LIN {X 0,Y 229.608,Z 438.992,A -85,B 0,C 180,E1 -19914.647,E2 -19914.647} C_VEL
LIN {X 0,Y 228.927,Z 425.746,A -85,B 0,C 180,E1 -19915.956,E2 -19915.956} C_VEL
LIN {X 0,Y 227.95,Z 410.113,A -85,B 0,C 180,E1 -19917.144,E2 -19917.144} C_VEL
LIN {X 0,Y 229.155,Z 402.055,A -85,B 0,C 180,E1 -19921.424,E2 -19921.424} C_VEL
LIN {X 0,Y 230.589,Z 394.783,A -85,B 0,C 180,E1 -19925.386,E2 -19925.386} C_VEL
LIN {X 0,Y 231.878,Z 388.889,A -85,B 0,C 180,E1 -19928.622,E2 -19928.622} C_VEL
LIN {X 0,Y 231.502,Z 385.409,A -85,B 0,C 180,E1 -19930.627,E2 -19930.627} C_VEL
LIN {X 0,Y 229.924,Z 377.597,A -85,B 0,C 180,E1 -19935.329,E2 -19935.329} C_VEL
LIN {X 0,Y 228.4,Z 369.835,A -85,B 0,C 180,E1 -19940.286,E2 -19940.286} C_VEL
LIN {X 0,Y 227.949,Z 367.157,A -85,B 0,C 180,E1 -19942.123,E2 -19942.123} C_VEL
LIN {X 0,Y 227.876,Z 367.099,A -85,B 0,C 180,E1 -19946.377,E2 -19946.377} C_VEL
LIN {X 0,Y 227.915,Z 367.092,A -85,B 0,C 180,E1 -19950.437,E2 -19950.437} C_VEL
LIN {X 0,Y 227.921,Z 367.093,A -85,B 0,C 180,E1 -19954.425,E2 -19954.425} C_VEL
LIN {X 0,Y 227.939,Z 367.087,A -85,B 0,C 180,E1 -19958.285,E2 -19958.285} C_VEL
LIN {X 0,Y 228.018,Z 367.079,A -85,B 0,C 180,E1 -19963.895,E2 -19963.895} C_VEL
LIN {X 0,Y 228.049,Z 367.073,A -85,B 0,C 180,E1 -19967.542,E2 -19967.542} C_VEL
LIN {X 0,Y 228.243,Z 367.054,A -85,B 0,C 180,E1 -19971.144,E2 -19971.144} C_VEL
LIN {X 0,Y 228.308,Z 367.048,A -85,B 0,C 180,E1 -19972.927,E2 -19972.927} C_VEL
LIN {X 0,Y 228.546,Z 367.013,A -85,B 0,C 180,E1 -19978.238,E2 -19978.238} C_VEL
LIN {X 0,Y 228.547,Z 367.014,A -85,B 0,C 180,E1 -19981.762,E2 -19981.762} C_VEL
LIN {X 0,Y 228.347,Z 367.04,A -85,B 0,C 180,E1 -19987.072,E2 -19987.072} C_VEL
LIN {X 0,Y 228.158,Z 367.066,A -85,B 0,C 180,E1 -19990.651,E2 -19990.651} C_VEL
LIN {X 0,Y 228.057,Z 367.074,A -85,B 0,C 180,E1 -19994.273,E2 -19994.273} C_VEL
LIN {X 0,Y 227.999,Z 367.083,A -85,B 0,C 180,E1 -19997.954,E2 -19997.954} C_VEL
LIN {X 0,Y 227.926,Z 367.091,A -85,B 0,C 180,E1 -20002.329,E2 -20002.329} C_VEL
LIN {X 0,Y 227.939,Z 367.092,A -85,B 0,C 180,E1 -20006.603,E2 -20006.603} C_VEL
LIN {X 0,Y 227.905,Z 367.095,A -85,B 0,C 180,E1 -20010.297,E2 -20010.297} C_VEL
LIN {X 0,Y 227.886,Z 367.097,A -85,B 0,C 180,E1 -20013.719,E2 -20013.719} C_VEL
LIN {X 0,Y 227.868,Z 367.099,A -85,B 0,C 180,E1 -20018.086,E2 -20018.086} C_VEL
LIN {X 0,Y 227.834,Z 367.107,A -85,B 0,C 180,E1 -20022.242,E2 -20022.242} C_VEL
LIN {X 0,Y 227.833,Z 367.102,A -85,B 0,C 180,E1 -20025.193,E2 -20025.193} C_VEL
LIN {X 0,Y 227.824,Z 367.105,A -85,B 0,C 180,E1 -20029.624,E2 -20029.624} C_VEL
LIN {X 0,Y 227.898,Z 367.095,A -85,B 0,C 180,E1 -20034.132,E2 -20034.132} C_VEL
LIN {X 0,Y 227.872,Z 367.1,A -85,B 0,C 180,E1 -20038.379,E2 -20038.379} C_VEL
LIN {X 0,Y 227.888,Z 367.094,A -85,B 0,C 180,E1 -20042.446,E2 -20042.446} C_VEL
LIN {X 0,Y 227.915,Z 367.094,A -85,B 0,C 180,E1 -20046.368,E2 -20046.368} C_VEL
LIN {X 0,Y 227.944,Z 367.088,A -85,B 0,C 180,E1 -20050.175,E2 -20050.175} C_VEL
LIN {X 0,Y 228.059,Z 367.078,A -85,B 0,C 180,E1 -20053.898,E2 -20053.898} C_VEL
LIN {X 0,Y 228.173,Z 367.06,A -85,B 0,C 180,E1 -20059.35,E2 -20059.35} C_VEL
LIN {X 0,Y 228.361,Z 367.038,A -85,B 0,C 180,E1 -20062.929,E2 -20062.929} C_VEL
LIN {X 0,Y 228.56,Z 367.013,A -85,B 0,C 180,E1 -20068.238,E2 -20068.238} C_VEL
LIN {X 0,Y 228.557,Z 367.014,A -85,B 0,C 180,E1 -20071.762,E2 -20071.762} C_VEL
LIN {X 0,Y 228.351,Z 367.038,A -85,B 0,C 180,E1 -20077.071,E2 -20077.071} C_VEL
LIN {X 0,Y 228.16,Z 367.062,A -85,B 0,C 180,E1 -20080.65,E2 -20080.65} C_VEL
LIN {X 0,Y 228.066,Z 367.074,A -85,B 0,C 180,E1 -20084.272,E2 -20084.272} C_VEL
LIN {X 0,Y 228.004,Z 367.083,A -85,B 0,C 180,E1 -20087.953,E2 -20087.953} C_VEL
LIN {X 0,Y 227.931,Z 367.092,A -85,B 0,C 180,E1 -20092.329,E2 -20092.329} C_VEL
LIN {X 0,Y 227.942,Z 367.09,A -85,B 0,C 180,E1 -20096.602,E2 -20096.602} C_VEL
LIN {X 0,Y 227.897,Z 367.097,A -85,B 0,C 180,E1 -20100.29,E2 -20100.29} C_VEL
LIN {X 0,Y 227.889,Z 367.098,A -85,B 0,C 180,E1 -20103.717,E2 -20103.717} C_VEL
LIN {X 0,Y 227.98,Z 367.279,A -85,B 0,C 180,E1 -20106.656,E2 -20106.656} C_VEL
LIN {X 0,Y 228.218,Z 368.301,A -85,B 0,C 180,E1 -20106.956,E2 -20106.956} C_VEL
LIN {X 0,Y 231.872,Z 380.761,A -85,B 0,C 180,E1 -20108.691,E2 -20108.691} C_VEL
LIN {X 0,Y 234.923,Z 392.226,A -85,B 0,C 180,E1 -20110.589,E2 -20110.589} C_VEL
LIN {X 0,Y 235.363,Z 394.934,A -85,B 0,C 180,E1 -20111.065,E2 -20111.065} C_VEL
LIN {X 0,Y 233.758,Z 406.693,A -85,B 0,C 180,E1 -20113.19,E2 -20113.19} C_VEL
LIN {X 0,Y 232.42,Z 416.268,A -85,B 0,C 180,E1 -20115.328,E2 -20115.328} C_VEL
LIN {X 0,Y 231,Z 425.883,A -85,B 0,C 180,E1 -20117.984,E2 -20117.984} C_VEL
LIN {X 0,Y 229.917,Z 433.61,A -85,B 0,C 180,E1 -20120.634,E2 -20120.634} C_VEL
LIN {X 0,Y 229.046,Z 440.448,A -85,B 0,C 180,E1 -20123.582,E2 -20123.582} C_VEL
LIN {X 0,Y 228.563,Z 445.529,A -85,B 0,C 180,E1 -20126.394,E2 -20126.394} C_VEL
LIN {X 0,Y 228.351,Z 449.786,A -85,B 0,C 180,E1 -20129.512,E2 -20129.512} C_VEL
LIN {X 0,Y 228.594,Z 453.024,A -85,B 0,C 180,E1 -20133.071,E2 -20133.071} C_VEL
LIN {X 0,Y 229.502,Z 454.674,A -85,B 0,C 180,E1 -20136.731,E2 -20136.731} C_VEL
LIN {X 0,Y 230.188,Z 454.837,A -85,B 0,C 180,E1 -20138.507,E2 -20138.507} C_VEL
LIN {X 0,Y 231.096,Z 454.553,A -85,B 0,C 180,E1 -20140.516,E2 -20140.516} C_VEL
LIN {X 0,Y 232.177,Z 453.845,A -85,B 0,C 180,E1 -20142.38,E2 -20142.38} C_VEL
LIN {X 0,Y 233.489,Z 452.509,A -85,B 0,C 180,E1 -20144.402,E2 -20144.402} C_VEL
LIN {X 0,Y 235.627,Z 449.858,A -85,B 0,C 180,E1 -20147.074,E2 -20147.074} C_VEL
LIN {X 0,Y 238.305,Z 445.922,A -85,B 0,C 180,E1 -20149.808,E2 -20149.808} C_VEL
LIN {X 0,Y 241.533,Z 440.446,A -85,B 0,C 180,E1 -20152.61,E2 -20152.61} C_VEL
LIN {X 0,Y 245.371,Z 433.011,A -85,B 0,C 180,E1 -20155.442,E2 -20155.442} C_VEL
LIN {X 0,Y 248.658,Z 425.827,A -85,B 0,C 180,E1 -20157.57,E2 -20157.57} C_VEL
LIN {X 0,Y 251.387,Z 419.09,A -85,B 0,C 180,E1 -20159.199,E2 -20159.199} C_VEL
LIN {X 0,Y 251.425,Z 416.583,A -85,B 0,C 180,E1 -20160,E2 -20160} C_VEL
LIN {X 0,Y 249.947,Z 407.014,A -85,B 0,C 180,E1 -20163.224,E2 -20163.224} C_VEL
LIN {X 0,Y 248.68,Z 402.352,A -85,B 0,C 180,E1 -20164.864,E2 -20164.864} C_VEL
LIN {X 0,Y 245.143,Z 393.716,A -85,B 0,C 180,E1 -20168.242,E2 -20168.242} C_VEL
LIN {X 0,Y 241.797,Z 387.198,A -85,B 0,C 180,E1 -20171.14,E2 -20171.14} C_VEL
LIN {X 0,Y 239.703,Z 383.456,A -85,B 0,C 180,E1 -20172.976,E2 -20172.976} C_VEL
LIN {X 0,Y 236.75,Z 379.72,A -85,B 0,C 180,E1 -20175.496,E2 -20175.496} C_VEL
LIN {X 0,Y 234.248,Z 377.714,A -85,B 0,C 180,E1 -20177.685,E2 -20177.685} C_VEL
LIN {X 0,Y 233.353,Z 376.567,A -85,B 0,C 180,E1 -20178.663,E2 -20178.663} C_VEL
LIN {X 0,Y 230.291,Z 375.175,A -85,B 0,C 180,E1 -20182.071,E2 -20182.071} C_VEL
LIN {X 0,Y 229.631,Z 374.388,A -85,B 0,C 180,E1 -20183.445,E2 -20183.445} C_VEL
LIN {X 0,Y 229.685,Z 374.739,A -85,B 0,C 180,E1 -20185.365,E2 -20185.365} C_VEL
LIN {X 0,Y 229.986,Z 375.936,A -85,B 0,C 180,E1 -20187.604,E2 -20187.604} C_VEL
LIN {X 0,Y 230.436,Z 378.369,A -85,B 0,C 180,E1 -20191.357,E2 -20191.357} C_VEL
LIN {X 0,Y 231.054,Z 381.457,A -85,B 0,C 180,E1 -20195.305,E2 -20195.305} C_VEL
LIN {X 0,Y 231.986,Z 385.695,A -85,B 0,C 180,E1 -20199.807,E2 -20199.807} C_VEL
LIN {X 0,Y 232.582,Z 388.031,A -85,B 0,C 180,E1 -20201.359,E2 -20201.359} C_VEL
LIN {X 0,Y 235.887,Z 395.137,A -85,B 0,C 180,E1 -20204.588,E2 -20204.588} C_VEL
LIN {X 0,Y 237.313,Z 397.724,A -85,B 0,C 180,E1 -20205.7,E2 -20205.7} C_VEL
LIN {X 0,Y 239.366,Z 402.878,A -85,B 0,C 180,E1 -20207.386,E2 -20207.386} C_VEL
LIN {X 0,Y 240.173,Z 404.323,A -85,B 0,C 180,E1 -20207.949,E2 -20207.949} C_VEL
LIN {X 0,Y 241.673,Z 410.353,A -85,B 0,C 180,E1 -20209.395,E2 -20209.395} C_VEL
LIN {X 0,Y 242.991,Z 419.215,A -85,B 0,C 180,E1 -20211.252,E2 -20211.252} C_VEL
LIN {X 0,Y 243.153,Z 423.985,A -85,B 0,C 180,E1 -20212.075,E2 -20212.075} C_VEL
LIN {X 0,Y 242.458,Z 429.111,A -85,B 0,C 180,E1 -20212.768,E2 -20212.768} C_VEL
LIN {X 0,Y 239.789,Z 439.501,A -85,B 0,C 180,E1 -20214.065,E2 -20214.065} C_VEL
LIN {X 0,Y 238.717,Z 444.414,A -85,B 0,C 180,E1 -20214.849,E2 -20214.849} C_VEL
LIN {X 0,Y 238.543,Z 445.927,A -85,B 0,C 180,E1 -20215.153,E2 -20215.153} C_VEL
LIN {X 0,Y 237.13,Z 458.322,A -85,B 0,C 180,E1 -20217.76,E2 -20217.76} C_VEL
LIN {X 0,Y 234.95,Z 468.801,A -85,B 0,C 180,E1 -20220.166,E2 -20220.166} C_VEL
LIN {X 0,Y 231.595,Z 479.491,A -85,B 0,C 180,E1 -20222.923,E2 -20222.923} C_VEL
LIN {X 0,Y 228.665,Z 487.706,A -85,B 0,C 180,E1 -20225.486,E2 -20225.486} C_VEL
LIN {X 0,Y 225.158,Z 495.637,A -85,B 0,C 180,E1 -20228.485,E2 -20228.485} C_VEL
LIN {X 0,Y 222.418,Z 502.006,A -85,B 0,C 180,E1 -20231.58,E2 -20231.58} C_VEL
LIN {X 0,Y 220.511,Z 507.656,A -85,B 0,C 180,E1 -20235.229,E2 -20235.229} C_VEL
LIN {X 0,Y 219.511,Z 511.634,A -85,B 0,C 180,E1 -20238.925,E2 -20238.925} C_VEL
LIN {X 0,Y 219.626,Z 514.192,A -85,B 0,C 180,E1 -20242.747,E2 -20242.747} C_VEL
LIN {X 0,Y 219.956,Z 514.809,A -85,B 0,C 180,E1 -20244.5,E2 -20244.5} C_VEL
LIN {X 0,Y 220.893,Z 514.907,A -85,B 0,C 180,E1 -20248.177,E2 -20248.177} C_VEL
LIN {X 0,Y 221.448,Z 514.346,A -85,B 0,C 180,E1 -20250,E2 -20250} C_VEL
LIN {X 0,Y 221.043,Z 513.169,A -85,B 0,C 180,E1 -20251.822,E2 -20251.822} C_VEL
LIN {X 0,Y 220.637,Z 510.508,A -85,B 0,C 180,E1 -20254.567,E2 -20254.567} C_VEL
LIN {X 0,Y 220.226,Z 506.669,A -85,B 0,C 180,E1 -20257.334,E2 -20257.334} C_VEL
LIN {X 0,Y 220.1,Z 501.587,A -85,B 0,C 180,E1 -20260.115,E2 -20260.115} C_VEL
LIN {X 0,Y 220.464,Z 495.155,A -85,B 0,C 180,E1 -20262.894,E2 -20262.894} C_VEL
LIN {X 0,Y 221.315,Z 487.153,A -85,B 0,C 180,E1 -20265.659,E2 -20265.659} C_VEL
LIN {X 0,Y 222.477,Z 479.009,A -85,B 0,C 180,E1 -20267.938,E2 -20267.938} C_VEL
LIN {X 0,Y 223.11,Z 473.256,A -85,B 0,C 180,E1 -20269.296,E2 -20269.296} C_VEL
LIN {X 0,Y 223.125,Z 462.474,A -85,B 0,C 180,E1 -20271.479,E2 -20271.479} C_VEL
LIN {X 0,Y 222.936,Z 451.084,A -85,B 0,C 180,E1 -20273.358,E2 -20273.358} C_VEL
LIN {X 0,Y 222.547,Z 438.854,A -85,B 0,C 180,E1 -20274.984,E2 -20274.984} C_VEL
LIN {X 0,Y 221.982,Z 426.264,A -85,B 0,C 180,E1 -20276.31,E2 -20276.31} C_VEL
LIN {X 0,Y 221.011,Z 410.739,A -85,B 0,C 180,E1 -20277.512,E2 -20277.512} C_VEL
LIN {X 0,Y 220.986,Z 408.993,A -85,B 0,C 180,E1 -20277.72,E2 -20277.72} C_VEL
LIN {X 0,Y 222.797,Z 398.631,A -85,B 0,C 180,E1 -20283.505,E2 -20283.505} C_VEL
LIN {X 0,Y 224.768,Z 389.696,A -85,B 0,C 180,E1 -20288.584,E2 -20288.584} C_VEL
LIN {X 0,Y 224.454,Z 386.287,A -85,B 0,C 180,E1 -20290.598,E2 -20290.598} C_VEL
LIN {X 0,Y 223.029,Z 379.316,A -85,B 0,C 180,E1 -20294.918,E2 -20294.918} C_VEL
LIN {X 0,Y 221.608,Z 372.183,A -85,B 0,C 180,E1 -20299.562,E2 -20299.562} C_VEL
LIN {X 0,Y 220.874,Z 368.016,A -85,B 0,C 180,E1 -20302.545,E2 -20302.545} C_VEL
LIN {X 0,Y 220.814,Z 367.981,A -85,B 0,C 180,E1 -20307.243,E2 -20307.243} C_VEL
LIN {X 0,Y 220.833,Z 367.976,A -85,B 0,C 180,E1 -20311.486,E2 -20311.486} C_VEL
LIN {X 0,Y 220.858,Z 367.972,A -85,B 0,C 180,E1 -20315.564,E2 -20315.564} C_VEL
LIN {X 0,Y 220.87,Z 367.971,A -85,B 0,C 180,E1 -20319.512,E2 -20319.512} C_VEL
LIN {X 0,Y 220.974,Z 367.958,A -85,B 0,C 180,E1 -20323.367,E2 -20323.367} C_VEL
LIN {X 0,Y 221.056,Z 367.947,A -85,B 0,C 180,E1 -20329.003,E2 -20329.003} C_VEL
LIN {X 0,Y 221.242,Z 367.927,A -85,B 0,C 180,E1 -20332.7,E2 -20332.7} C_VEL
LIN {X 0,Y 221.504,Z 367.89,A -85,B 0,C 180,E1 -20338.182,E2 -20338.182} C_VEL
LIN {X 0,Y 221.505,Z 367.891,A -85,B 0,C 180,E1 -20341.818,E2 -20341.818} C_VEL
LIN {X 0,Y 221.283,Z 367.919,A -85,B 0,C 180,E1 -20347.299,E2 -20347.299} C_VEL
LIN {X 0,Y 221.107,Z 367.942,A -85,B 0,C 180,E1 -20350.994,E2 -20350.994} C_VEL
LIN {X 0,Y 221.011,Z 367.957,A -85,B 0,C 180,E1 -20356.63,E2 -20356.63} C_VEL
LIN {X 0,Y 220.888,Z 367.969,A -85,B 0,C 180,E1 -20360.487,E2 -20360.487} C_VEL
LIN {X 0,Y 220.863,Z 367.974,A -85,B 0,C 180,E1 -20364.435,E2 -20364.435} C_VEL
LIN {X 0,Y 220.833,Z 367.976,A -85,B 0,C 180,E1 -20368.514,E2 -20368.514} C_VEL
LIN {X 0,Y 220.821,Z 367.978,A -85,B 0,C 180,E1 -20372.755,E2 -20372.755} C_VEL
LIN {X 0,Y 220.836,Z 367.973,A -85,B 0,C 180,E1 -20377.289,E2 -20377.289} C_VEL
LIN {X 0,Y 220.835,Z 367.977,A -85,B 0,C 180,E1 -20380.202,E2 -20380.202} C_VEL
LIN {X 0,Y 220.777,Z 367.983,A -85,B 0,C 180,E1 -20384.453,E2 -20384.453} C_VEL
LIN {X 0,Y 220.768,Z 367.984,A -85,B 0,C 180,E1 -20388.048,E2 -20388.048} C_VEL
LIN {X 0,Y 220.823,Z 367.975,A -85,B 0,C 180,E1 -20392.794,E2 -20392.794} C_VEL
LIN {X 0,Y 220.823,Z 367.976,A -85,B 0,C 180,E1 -20397.246,E2 -20397.246} C_VEL
LIN {X 0,Y 220.838,Z 367.975,A -85,B 0,C 180,E1 -20401.487,E2 -20401.487} C_VEL
LIN {X 0,Y 220.868,Z 367.972,A -85,B 0,C 180,E1 -20405.566,E2 -20405.566} C_VEL
LIN {X 0,Y 220.894,Z 367.969,A -85,B 0,C 180,E1 -20409.515,E2 -20409.515} C_VEL
LIN {X 0,Y 221.018,Z 367.952,A -85,B 0,C 180,E1 -20413.371,E2 -20413.371} C_VEL
LIN {X 0,Y 221.118,Z 367.938,A -85,B 0,C 180,E1 -20419.006,E2 -20419.006} C_VEL
LIN {X 0,Y 221.314,Z 367.915,A -85,B 0,C 180,E1 -20422.703,E2 -20422.703} C_VEL
LIN {X 0,Y 221.517,Z 367.89,A -85,B 0,C 180,E1 -20428.182,E2 -20428.182} C_VEL
LIN {X 0,Y 221.515,Z 367.891,A -85,B 0,C 180,E1 -20431.818,E2 -20431.818} C_VEL
LIN {X 0,Y 221.286,Z 367.919,A -85,B 0,C 180,E1 -20437.298,E2 -20437.298} C_VEL
LIN {X 0,Y 221.108,Z 367.942,A -85,B 0,C 180,E1 -20440.994,E2 -20440.994} C_VEL
LIN {X 0,Y 221.018,Z 367.952,A -85,B 0,C 180,E1 -20446.629,E2 -20446.629} C_VEL
LIN {X 0,Y 220.894,Z 367.968,A -85,B 0,C 180,E1 -20450.485,E2 -20450.485} C_VEL
LIN {X 0,Y 220.868,Z 367.971,A -85,B 0,C 180,E1 -20454.434,E2 -20454.434} C_VEL
LIN {X 0,Y 220.827,Z 367.977,A -85,B 0,C 180,E1 -20458.514,E2 -20458.514} C_VEL
LIN {X 0,Y 220.822,Z 367.979,A -85,B 0,C 180,E1 -20462.754,E2 -20462.754} C_VEL
LIN {X 0,Y 220.938,Z 368.197,A -85,B 0,C 180,E1 -20466.189,E2 -20466.189} C_VEL
LIN {X 0,Y 221.315,Z 369.606,A -85,B 0,C 180,E1 -20466.541,E2 -20466.541} C_VEL
LIN {X 0,Y 225.032,Z 382.472,A -85,B 0,C 180,E1 -20468.391,E2 -20468.391} C_VEL
LIN {X 0,Y 228.05,Z 393.725,A -85,B 0,C 180,E1 -20470.328,E2 -20470.328} C_VEL
LIN {X 0,Y 228.436,Z 396.031,A -85,B 0,C 180,E1 -20470.746,E2 -20470.746} C_VEL
LIN {X 0,Y 227,Z 406.259,A -85,B 0,C 180,E1 -20472.623,E2 -20472.623} C_VEL
LIN {X 0,Y 225.346,Z 417.549,A -85,B 0,C 180,E1 -20475.199,E2 -20475.199} C_VEL
LIN {X 0,Y 224.07,Z 426.024,A -85,B 0,C 180,E1 -20477.596,E2 -20477.596} C_VEL
LIN {X 0,Y 222.908,Z 434.092,A -85,B 0,C 180,E1 -20480.41,E2 -20480.41} C_VEL
LIN {X 0,Y 222.102,Z 440.214,A -85,B 0,C 180,E1 -20483.043,E2 -20483.043} C_VEL
LIN {X 0,Y 221.481,Z 446.408,A -85,B 0,C 180,E1 -20486.444,E2 -20486.444} C_VEL
LIN {X 0,Y 221.305,Z 450.496,A -85,B 0,C 180,E1 -20489.462,E2 -20489.462} C_VEL
LIN {X 0,Y 221.488,Z 453.578,A -85,B 0,C 180,E1 -20492.678,E2 -20492.678} C_VEL
LIN {X 0,Y 222.372,Z 455.557,A -85,B 0,C 180,E1 -20496.422,E2 -20496.422} C_VEL
LIN {X 0,Y 223.72,Z 455.93,A -85,B 0,C 180,E1 -20499.784,E2 -20499.784} C_VEL
LIN {X 0,Y 224.754,Z 455.531,A -85,B 0,C 180,E1 -20501.778,E2 -20501.778} C_VEL
LIN {X 0,Y 226.352,Z 454.314,A -85,B 0,C 180,E1 -20504.258,E2 -20504.258} C_VEL
LIN {X 0,Y 229.023,Z 451.371,A -85,B 0,C 180,E1 -20507.596,E2 -20507.596} C_VEL
LIN {X 0,Y 231.875,Z 447.588,A -85,B 0,C 180,E1 -20510.404,E2 -20510.404} C_VEL
LIN {X 0,Y 235.101,Z 442.579,A -85,B 0,C 180,E1 -20513.133,E2 -20513.133} C_VEL
LIN {X 0,Y 238.723,Z 436.177,A -85,B 0,C 180,E1 -20515.768,E2 -20515.768} C_VEL
LIN {X 0,Y 242.764,Z 428.059,A -85,B 0,C 180,E1 -20518.341,E2 -20518.341} C_VEL
LIN {X 0,Y 245.655,Z 421.564,A -85,B 0,C 180,E1 -20520,E2 -20520} C_VEL
LIN {X 0,Y 245.225,Z 415.957,A -85,B 0,C 180,E1 -20522.053,E2 -20522.053} C_VEL
LIN {X 0,Y 244.303,Z 409.245,A -85,B 0,C 180,E1 -20524.465,E2 -20524.465} C_VEL
LIN {X 0,Y 242.566,Z 403.762,A -85,B 0,C 180,E1 -20526.655,E2 -20526.655} C_VEL
LIN {X 0,Y 239.933,Z 396.884,A -85,B 0,C 180,E1 -20529.61,E2 -20529.61} C_VEL
LIN {X 0,Y 236.466,Z 389.951,A -85,B 0,C 180,E1 -20533.156,E2 -20533.156} C_VEL
LIN {X 0,Y 233.769,Z 386.071,A -85,B 0,C 180,E1 -20535.841,E2 -20535.841} C_VEL
LIN {X 0,Y 230.623,Z 383.152,A -85,B 0,C 180,E1 -20539.149,E2 -20539.149} C_VEL
LIN {X 0,Y 227.995,Z 381.679,A -85,B 0,C 180,E1 -20542.633,E2 -20542.633} C_VEL
LIN {X 0,Y 227.528,Z 381.149,A -85,B 0,C 180,E1 -20543.675,E2 -20543.675} C_VEL
LIN {X 0,Y 226.051,Z 381.62,A -85,B 0,C 180,E1 -20547.105,E2 -20547.105} C_VEL
LIN {X 0,Y 225.556,Z 383.422,A -85,B 0,C 180,E1 -20551.095,E2 -20551.095} C_VEL
LIN {X 0,Y 226.222,Z 386.236,A -85,B 0,C 180,E1 -20554.588,E2 -20554.588} C_VEL
LIN {X 0,Y 228.937,Z 391.93,A -85,B 0,C 180,E1 -20559.427,E2 -20559.427} C_VEL
LIN {X 0,Y 230.112,Z 394.682,A -85,B 0,C 180,E1 -20560.976,E2 -20560.976} C_VEL
LIN {X 0,Y 232.854,Z 401.033,A -85,B 0,C 180,E1 -20563.963,E2 -20563.963} C_VEL
LIN {X 0,Y 233.668,Z 402.418,A -85,B 0,C 180,E1 -20564.675,E2 -20564.675} C_VEL
LIN {X 0,Y 235.763,Z 408.322,A -85,B 0,C 180,E1 -20566.717,E2 -20566.717} C_VEL
LIN {X 0,Y 236.66,Z 410.544,A -85,B 0,C 180,E1 -20567.509,E2 -20567.509} C_VEL
LIN {X 0,Y 237.395,Z 415.062,A -85,B 0,C 180,E1 -20568.6,E2 -20568.6} C_VEL
LIN {X 0,Y 238.328,Z 423.701,A -85,B 0,C 180,E1 -20570.517,E2 -20570.517} C_VEL
LIN {X 0,Y 238.854,Z 436.554,A -85,B 0,C 180,E1 -20573.205,E2 -20573.205} C_VEL
LIN {X 0,Y 238.543,Z 445.927,A -85,B 0,C 180,E1 -20575.153,E2 -20575.153} C_VEL
LIN {X 0,Y 237.596,Z 450.708,A -85,B 0,C 180,E1 -20576.014,E2 -20576.014} C_VEL
LIN {X 0,Y 235.73,Z 455.509,A -85,B 0,C 180,E1 -20576.759,E2 -20576.759} C_VEL
LIN {X 0,Y 231.021,Z 464.66,A -85,B 0,C 180,E1 -20578.239,E2 -20578.239} C_VEL
LIN {X 0,Y 229.077,Z 468.943,A -85,B 0,C 180,E1 -20579.133,E2 -20579.133} C_VEL
LIN {X 0,Y 228.619,Z 470.288,A -85,B 0,C 180,E1 -20579.468,E2 -20579.468} C_VEL
LIN {X 0,Y 225.282,Z 479.825,A -85,B 0,C 180,E1 -20582.1,E2 -20582.1} C_VEL
LIN {X 0,Y 221.657,Z 488.946,A -85,B 0,C 180,E1 -20585.159,E2 -20585.159} C_VEL
LIN {X 0,Y 218.079,Z 496.39,A -85,B 0,C 180,E1 -20588.247,E2 -20588.247} C_VEL
LIN {X 0,Y 215.056,Z 503.063,A -85,B 0,C 180,E1 -20591.914,E2 -20591.914} C_VEL
LIN {X 0,Y 213.215,Z 508.098,A -85,B 0,C 180,E1 -20595.688,E2 -20595.688} C_VEL
LIN {X 0,Y 212.502,Z 510.799,A -85,B 0,C 180,E1 -20598.555,E2 -20598.555} C_VEL
LIN {X 0,Y 212.537,Z 513.13,A -85,B 0,C 180,E1 -20602.4,E2 -20602.4} C_VEL
LIN {X 0,Y 212.886,Z 513.711,A -85,B 0,C 180,E1 -20604.316,E2 -20604.316} C_VEL
LIN {X 0,Y 213.845,Z 513.703,A -85,B 0,C 180,E1 -20608.117,E2 -20608.117} C_VEL
LIN {X 0,Y 214.431,Z 513.093,A -85,B 0,C 180,E1 -20610,E2 -20610} C_VEL
LIN {X 0,Y 214.039,Z 511.812,A -85,B 0,C 180,E1 -20611.882,E2 -20611.882} C_VEL
LIN {X 0,Y 213.613,Z 509.022,A -85,B 0,C 180,E1 -20614.718,E2 -20614.718} C_VEL
LIN {X 0,Y 213.175,Z 505.032,A -85,B 0,C 180,E1 -20617.578,E2 -20617.578} C_VEL
LIN {X 0,Y 213.166,Z 498.831,A -85,B 0,C 180,E1 -20620.928,E2 -20620.928} C_VEL
LIN {X 0,Y 213.61,Z 491.961,A -85,B 0,C 180,E1 -20623.8,E2 -20623.8} C_VEL
LIN {X 0,Y 214.676,Z 483.403,A -85,B 0,C 180,E1 -20626.645,E2 -20626.645} C_VEL
LIN {X 0,Y 215.976,Z 474.691,A -85,B 0,C 180,E1 -20628.99,E2 -20628.99} C_VEL
LIN {X 0,Y 216.065,Z 464.592,A -85,B 0,C 180,E1 -20631.214,E2 -20631.214} C_VEL
LIN {X 0,Y 215.905,Z 452.698,A -85,B 0,C 180,E1 -20633.351,E2 -20633.351} C_VEL
LIN {X 0,Y 215.644,Z 440.924,A -85,B 0,C 180,E1 -20635.066,E2 -20635.066} C_VEL
LIN {X 0,Y 215.114,Z 427.854,A -85,B 0,C 180,E1 -20636.563,E2 -20636.563} C_VEL
LIN {X 0,Y 214.351,Z 414.249,A -85,B 0,C 180,E1 -20637.746,E2 -20637.746} C_VEL
LIN {X 0,Y 214.006,Z 408.243,A -85,B 0,C 180,E1 -20638.214,E2 -20638.214} C_VEL
LIN {X 0,Y 215.331,Z 400.48,A -85,B 0,C 180,E1 -20642.647,E2 -20642.647} C_VEL
LIN {X 0,Y 217.355,Z 391.513,A -85,B 0,C 180,E1 -20647.903,E2 -20647.903} C_VEL
LIN {X 0,Y 217.723,Z 389.305,A -85,B 0,C 180,E1 -20649.221,E2 -20649.221} C_VEL
LIN {X 0,Y 216.625,Z 383.378,A -85,B 0,C 180,E1 -20652.944,E2 -20652.944} C_VEL
LIN {X 0,Y 215.095,Z 375.852,A -85,B 0,C 180,E1 -20657.885,E2 -20657.885} C_VEL
LIN {X 0,Y 213.83,Z 368.918,A -85,B 0,C 180,E1 -20662.769,E2 -20662.769} C_VEL
LIN {X 0,Y 213.754,Z 368.858,A -85,B 0,C 180,E1 -20666.017,E2 -20666.017} C_VEL
LIN {X 0,Y 213.777,Z 368.853,A -85,B 0,C 180,E1 -20670.453,E2 -20670.453} C_VEL
LIN {X 0,Y 213.794,Z 368.853,A -85,B 0,C 180,E1 -20674.701,E2 -20674.701} C_VEL
LIN {X 0,Y 213.792,Z 368.851,A -85,B 0,C 180,E1 -20678.801,E2 -20678.801} C_VEL
LIN {X 0,Y 213.888,Z 368.843,A -85,B 0,C 180,E1 -20682.799,E2 -20682.799} C_VEL
LIN {X 0,Y 213.929,Z 368.831,A -85,B 0,C 180,E1 -20686.705,E2 -20686.705} C_VEL
LIN {X 0,Y 214.12,Z 368.811,A -85,B 0,C 180,E1 -20690.554,E2 -20690.554} C_VEL
LIN {X 0,Y 214.087,Z 368.816,A -85,B 0,C 180,E1 -20694.348,E2 -20694.348} C_VEL
LIN {X 0,Y 214.437,Z 368.77,A -85,B 0,C 180,E1 -20698.122,E2 -20698.122} C_VEL
LIN {X 0,Y 214.544,Z 368.758,A -85,B 0,C 180,E1 -20700,E2 -20700} C_VEL
LIN {X 0,Y 214.438,Z 368.772,A -85,B 0,C 180,E1 -20701.878,E2 -20701.878} C_VEL
LIN {X 0,Y 214.221,Z 368.798,A -85,B 0,C 180,E1 -20707.541,E2 -20707.541} C_VEL
LIN {X 0,Y 214.04,Z 368.821,A -85,B 0,C 180,E1 -20711.362,E2 -20711.362} C_VEL
LIN {X 0,Y 213.927,Z 368.835,A -85,B 0,C 180,E1 -20715.237,E2 -20715.237} C_VEL
LIN {X 0,Y 213.835,Z 368.847,A -85,B 0,C 180,E1 -20719.188,E2 -20719.188} C_VEL
LIN {X 0,Y 213.843,Z 368.845,A -85,B 0,C 180,E1 -20723.227,E2 -20723.227} C_VEL
LIN {X 0,Y 213.826,Z 368.848,A -85,B 0,C 180,E1 -20727.45,E2 -20727.45} C_VEL
LIN {X 0,Y 213.776,Z 368.853,A -85,B 0,C 180,E1 -20731.736,E2 -20731.736} C_VEL
LIN {X 0,Y 213.751,Z 368.859,A -85,B 0,C 180,E1 -20736.287,E2 -20736.287} C_VEL
LIN {X 0,Y 213.75,Z 368.858,A -85,B 0,C 180,E1 -20740.869,E2 -20740.869} C_VEL
LIN {X 0,Y 213.746,Z 368.859,A -85,B 0,C 180,E1 -20743.669,E2 -20743.669} C_VEL
LIN {X 0,Y 213.71,Z 368.862,A -85,B 0,C 180,E1 -20748.876,E2 -20748.876} C_VEL
LIN {X 0,Y 213.747,Z 368.858,A -85,B 0,C 180,E1 -20753.713,E2 -20753.713} C_VEL
LIN {X 0,Y 213.779,Z 368.856,A -85,B 0,C 180,E1 -20758.265,E2 -20758.265} C_VEL
LIN {X 0,Y 213.826,Z 368.845,A -85,B 0,C 180,E1 -20762.604,E2 -20762.604} C_VEL
LIN {X 0,Y 213.853,Z 368.845,A -85,B 0,C 180,E1 -20766.953,E2 -20766.953} C_VEL
LIN {X 0,Y 213.945,Z 368.832,A -85,B 0,C 180,E1 -20772.804,E2 -20772.804} C_VEL
LIN {X 0,Y 213.982,Z 368.828,A -85,B 0,C 180,E1 -20776.709,E2 -20776.709} C_VEL
LIN {X 0,Y 214.198,Z 368.8,A -85,B 0,C 180,E1 -20780.558,E2 -20780.558} C_VEL
LIN {X 0,Y 214.25,Z 368.796,A -85,B 0,C 180,E1 -20782.461,E2 -20782.461} C_VEL
LIN {X 0,Y 214.451,Z 368.771,A -85,B 0,C 180,E1 -20788.122,E2 -20788.122} C_VEL
LIN {X 0,Y 214.557,Z 368.758,A -85,B 0,C 180,E1 -20790,E2 -20790} C_VEL
LIN {X 0,Y 214.449,Z 368.771,A -85,B 0,C 180,E1 -20791.878,E2 -20791.878} C_VEL
LIN {X 0,Y 214.224,Z 368.801,A -85,B 0,C 180,E1 -20797.54,E2 -20797.54} C_VEL
LIN {X 0,Y 214.025,Z 368.823,A -85,B 0,C 180,E1 -20801.363,E2 -20801.363} C_VEL
LIN {X 0,Y 213.936,Z 368.838,A -85,B 0,C 180,E1 -20805.236,E2 -20805.236} C_VEL
LIN {X 0,Y 213.869,Z 368.846,A -85,B 0,C 180,E1 -20809.184,E2 -20809.184} C_VEL
LIN {X 0,Y 213.848,Z 368.848,A -85,B 0,C 180,E1 -20813.226,E2 -20813.226} C_VEL
LIN {X 0,Y 213.829,Z 368.85,A -85,B 0,C 180,E1 -20817.449,E2 -20817.449} C_VEL
LIN {X 0,Y 213.769,Z 368.858,A -85,B 0,C 180,E1 -20821.736,E2 -20821.736} C_VEL
LIN {X 0,Y 213.868,Z 369.06,A -85,B 0,C 180,E1 -20825.672,E2 -20825.672} C_VEL
LIN {X 0,Y 214.114,Z 370.059,A -85,B 0,C 180,E1 -20825.978,E2 -20825.978} C_VEL
LIN {X 0,Y 217.996,Z 383.346,A -85,B 0,C 180,E1 -20827.965,E2 -20827.965} C_VEL
LIN {X 0,Y 221.115,Z 395.078,A -85,B 0,C 180,E1 -20830.057,E2 -20830.057} C_VEL
LIN {X 0,Y 221.478,Z 396.873,A -85,B 0,C 180,E1 -20830.397,E2 -20830.397} C_VEL
LIN {X 0,Y 219.996,Z 407.293,A -85,B 0,C 180,E1 -20832.369,E2 -20832.369} C_VEL
LIN {X 0,Y 218.367,Z 418.19,A -85,B 0,C 180,E1 -20834.923,E2 -20834.923} C_VEL
LIN {X 0,Y 216.859,Z 427.936,A -85,B 0,C 180,E1 -20837.786,E2 -20837.786} C_VEL
LIN {X 0,Y 215.729,Z 435.546,A -85,B 0,C 180,E1 -20840.559,E2 -20840.559} C_VEL
LIN {X 0,Y 214.964,Z 441.792,A -85,B 0,C 180,E1 -20843.369,E2 -20843.369} C_VEL
LIN {X 0,Y 214.444,Z 446.742,A -85,B 0,C 180,E1 -20846.142,E2 -20846.142} C_VEL
LIN {X 0,Y 214.241,Z 451.316,A -85,B 0,C 180,E1 -20849.52,E2 -20849.52} C_VEL
LIN {X 0,Y 214.444,Z 454.361,A -85,B 0,C 180,E1 -20852.689,E2 -20852.689} C_VEL
LIN {X 0,Y 215.222,Z 456.387,A -85,B 0,C 180,E1 -20856.107,E2 -20856.107} C_VEL
LIN {X 0,Y 216.808,Z 457.086,A -85,B 0,C 180,E1 -20860.057,E2 -20860.057} C_VEL
LIN {X 0,Y 219.194,Z 455.989,A -85,B 0,C 180,E1 -20864.125,E2 -20864.125} C_VEL
LIN {X 0,Y 221.572,Z 453.852,A -85,B 0,C 180,E1 -20867.172,E2 -20867.172} C_VEL
LIN {X 0,Y 224.414,Z 450.61,A -85,B 0,C 180,E1 -20870.082,E2 -20870.082} C_VEL
LIN {X 0,Y 227.74,Z 446.143,A -85,B 0,C 180,E1 -20872.909,E2 -20872.909} C_VEL
LIN {X 0,Y 231.389,Z 440.447,A -85,B 0,C 180,E1 -20875.646,E2 -20875.646} C_VEL
LIN {X 0,Y 235.506,Z 433.15,A -85,B 0,C 180,E1 -20878.29,E2 -20878.29} C_VEL
LIN {X 0,Y 239.494,Z 425.126,A -85,B 0,C 180,E1 -20880.563,E2 -20880.563} C_VEL
LIN {X 0,Y 239.894,Z 424.111,A -85,B 0,C 180,E1 -20880.839,E2 -20880.839} C_VEL
LIN {X 0,Y 239.375,Z 415.707,A -85,B 0,C 180,E1 -20884.125,E2 -20884.125} C_VEL
LIN {X 0,Y 238.315,Z 410.413,A -85,B 0,C 180,E1 -20886.314,E2 -20886.314} C_VEL
LIN {X 0,Y 235.474,Z 401.735,A -85,B 0,C 180,E1 -20890.316,E2 -20890.316} C_VEL
LIN {X 0,Y 232.489,Z 395.187,A -85,B 0,C 180,E1 -20893.995,E2 -20893.995} C_VEL
LIN {X 0,Y 230.833,Z 392.59,A -85,B 0,C 180,E1 -20895.904,E2 -20895.904} C_VEL
LIN {X 0,Y 227.515,Z 389.609,A -85,B 0,C 180,E1 -20899.864,E2 -20899.864} C_VEL
LIN {X 0,Y 225.208,Z 387.932,A -85,B 0,C 180,E1 -20903.934,E2 -20903.934} C_VEL
LIN {X 0,Y 224.273,Z 388.149,A -85,B 0,C 180,E1 -20906.022,E2 -20906.022} C_VEL
LIN {X 0,Y 223.526,Z 389.789,A -85,B 0,C 180,E1 -20910.203,E2 -20910.203} C_VEL
LIN {X 0,Y 223.613,Z 391.144,A -85,B 0,C 180,E1 -20912.296,E2 -20912.296} C_VEL
LIN {X 0,Y 224.873,Z 395.2,A -85,B 0,C 180,E1 -20916.428,E2 -20916.428} C_VEL
LIN {X 0,Y 226.906,Z 399.457,A -85,B 0,C 180,E1 -20919.745,E2 -20919.745} C_VEL
LIN {X 0,Y 229.482,Z 406.676,A -85,B 0,C 180,E1 -20923.268,E2 -20923.268} C_VEL
LIN {X 0,Y 230.166,Z 407.946,A -85,B 0,C 180,E1 -20923.937,E2 -20923.937} C_VEL
LIN {X 0,Y 231.606,Z 412.88,A -85,B 0,C 180,E1 -20925.741,E2 -20925.741} C_VEL
LIN {X 0,Y 232.46,Z 414.755,A -85,B 0,C 180,E1 -20926.519,E2 -20926.519} C_VEL
LIN {X 0,Y 233.039,Z 419.357,A -85,B 0,C 180,E1 -20927.725,E2 -20927.725} C_VEL
LIN {X 0,Y 233.62,Z 430.225,A -85,B 0,C 180,E1 -20930.265,E2 -20930.265} C_VEL
LIN {X 0,Y 233.337,Z 442.371,A -85,B 0,C 180,E1 -20932.96,E2 -20932.96} C_VEL
LIN {X 0,Y 232.389,Z 452.338,A -85,B 0,C 180,E1 -20935.179,E2 -20935.179} C_VEL
LIN {X 0,Y 230.42,Z 463.364,A -85,B 0,C 180,E1 -20937.741,E2 -20937.741} C_VEL
LIN {X 0,Y 228.619,Z 470.288,A -85,B 0,C 180,E1 -20939.468,E2 -20939.468} C_VEL
LIN {X 0,Y 226.793,Z 474.361,A -85,B 0,C 180,E1 -20940.448,E2 -20940.448} C_VEL
LIN {X 0,Y 221.999,Z 480.777,A -85,B 0,C 180,E1 -20941.944,E2 -20941.944} C_VEL
LIN {X 0,Y 216.933,Z 486.661,A -85,B 0,C 180,E1 -20943.572,E2 -20943.572} C_VEL
LIN {X 0,Y 214.728,Z 489.911,A -85,B 0,C 180,E1 -20944.748,E2 -20944.748} C_VEL
LIN {X 0,Y 211.471,Z 496.127,A -85,B 0,C 180,E1 -20947.531,E2 -20947.531} C_VEL
LIN {X 0,Y 208.199,Z 502.664,A -85,B 0,C 180,E1 -20951.363,E2 -20951.363} C_VEL
LIN {X 0,Y 206.288,Z 507.358,A -85,B 0,C 180,E1 -20955.196,E2 -20955.196} C_VEL
LIN {X 0,Y 205.493,Z 509.963,A -85,B 0,C 180,E1 -20958.159,E2 -20958.159} C_VEL
LIN {X 0,Y 205.456,Z 512.095,A -85,B 0,C 180,E1 -20962.136,E2 -20962.136} C_VEL
LIN {X 0,Y 205.818,Z 512.622,A -85,B 0,C 180,E1 -20964.12,E2 -20964.12} C_VEL
LIN {X 0,Y 206.824,Z 512.483,A -85,B 0,C 180,E1 -20968.053,E2 -20968.053} C_VEL
LIN {X 0,Y 207.434,Z 511.762,A -85,B 0,C 180,E1 -20970,E2 -20970} C_VEL
LIN {X 0,Y 207.031,Z 510.407,A -85,B 0,C 180,E1 -20971.945,E2 -20971.945} C_VEL
LIN {X 0,Y 206.584,Z 507.484,A -85,B 0,C 180,E1 -20974.879,E2 -20974.879} C_VEL
LIN {X 0,Y 206.128,Z 503.352,A -85,B 0,C 180,E1 -20977.838,E2 -20977.838} C_VEL
LIN {X 0,Y 206.128,Z 497.992,A -85,B 0,C 180,E1 -20980.808,E2 -20980.808} C_VEL
LIN {X 0,Y 206.554,Z 491.21,A -85,B 0,C 180,E1 -20983.778,E2 -20983.778} C_VEL
LIN {X 0,Y 207.627,Z 482.742,A -85,B 0,C 180,E1 -20986.721,E2 -20986.721} C_VEL
LIN {X 0,Y 208.902,Z 474.1,A -85,B 0,C 180,E1 -20989.148,E2 -20989.148} C_VEL
LIN {X 0,Y 208.979,Z 464.104,A -85,B 0,C 180,E1 -20991.452,E2 -20991.452} C_VEL
LIN {X 0,Y 208.846,Z 452.934,A -85,B 0,C 180,E1 -20993.553,E2 -20993.553} C_VEL
LIN {X 0,Y 208.603,Z 440.993,A -85,B 0,C 180,E1 -20995.384,E2 -20995.384} C_VEL
LIN {X 0,Y 208.132,Z 427.977,A -85,B 0,C 180,E1 -20996.959,E2 -20996.959} C_VEL
LIN {X 0,Y 207.367,Z 413.677,A -85,B 0,C 180,E1 -20998.263,E2 -20998.263} C_VEL
LIN {X 0,Y 207.055,Z 407.381,A -85,B 0,C 180,E1 -20998.787,E2 -20998.787} C_VEL
LIN {X 0,Y 207.523,Z 404.245,A -85,B 0,C 180,E1 -21000.529,E2 -21000.529} C_VEL
LIN {X 0,Y 209.335,Z 395.822,A -85,B 0,C 180,E1 -21005.643,E2 -21005.643} C_VEL
LIN {X 0,Y 210.333,Z 391.683,A -85,B 0,C 180,E1 -21008.18,E2 -21008.18} C_VEL
LIN {X 0,Y 210.524,Z 389.004,A -85,B 0,C 180,E1 -21009.841,E2 -21009.841} C_VEL
LIN {X 0,Y 209.337,Z 382.935,A -85,B 0,C 180,E1 -21013.797,E2 -21013.797} C_VEL
LIN {X 0,Y 207.784,Z 375.415,A -85,B 0,C 180,E1 -21018.976,E2 -21018.976} C_VEL
LIN {X 0,Y 206.776,Z 369.788,A -85,B 0,C 180,E1 -21023.123,E2 -21023.123} C_VEL
LIN {X 0,Y 206.723,Z 369.733,A -85,B 0,C 180,E1 -21028.202,E2 -21028.202} C_VEL
LIN {X 0,Y 206.763,Z 369.727,A -85,B 0,C 180,E1 -21032.096,E2 -21032.096} C_VEL
LIN {X 0,Y 206.75,Z 369.729,A -85,B 0,C 180,E1 -21036.604,E2 -21036.604} C_VEL
LIN {X 0,Y 206.821,Z 369.721,A -85,B 0,C 180,E1 -21042.192,E2 -21042.192} C_VEL
LIN {X 0,Y 206.87,Z 369.709,A -85,B 0,C 180,E1 -21046.242,E2 -21046.242} C_VEL
LIN {X 0,Y 207.067,Z 369.688,A -85,B 0,C 180,E1 -21050.229,E2 -21050.229} C_VEL
LIN {X 0,Y 207.048,Z 369.692,A -85,B 0,C 180,E1 -21054.155,E2 -21054.155} C_VEL
LIN {X 0,Y 207.374,Z 369.65,A -85,B 0,C 180,E1 -21058.058,E2 -21058.058} C_VEL
LIN {X 0,Y 207.509,Z 369.635,A -85,B 0,C 180,E1 -21060,E2 -21060} C_VEL
LIN {X 0,Y 207.375,Z 369.652,A -85,B 0,C 180,E1 -21061.942,E2 -21061.942} C_VEL
LIN {X 0,Y 207.162,Z 369.678,A -85,B 0,C 180,E1 -21067.799,E2 -21067.799} C_VEL
LIN {X 0,Y 206.977,Z 369.7,A -85,B 0,C 180,E1 -21071.755,E2 -21071.755} C_VEL
LIN {X 0,Y 206.861,Z 369.715,A -85,B 0,C 180,E1 -21075.771,E2 -21075.771} C_VEL
LIN {X 0,Y 206.779,Z 369.725,A -85,B 0,C 180,E1 -21079.87,E2 -21079.87} C_VEL
LIN {X 0,Y 206.76,Z 369.728,A -85,B 0,C 180,E1 -21084.073,E2 -21084.073} C_VEL
LIN {X 0,Y 206.741,Z 369.731,A -85,B 0,C 180,E1 -21088.419,E2 -21088.419} C_VEL
LIN {X 0,Y 206.706,Z 369.736,A -85,B 0,C 180,E1 -21092.956,E2 -21092.956} C_VEL
LIN {X 0,Y 206.721,Z 369.732,A -85,B 0,C 180,E1 -21097.731,E2 -21097.731} C_VEL
LIN {X 0,Y 206.669,Z 369.74,A -85,B 0,C 180,E1 -21101.573,E2 -21101.573} C_VEL
LIN {X 0,Y 206.641,Z 369.742,A -85,B 0,C 180,E1 -21105.58,E2 -21105.58} C_VEL
LIN {X 0,Y 206.662,Z 369.742,A -85,B 0,C 180,E1 -21109.75,E2 -21109.75} C_VEL
LIN {X 0,Y 206.731,Z 369.729,A -85,B 0,C 180,E1 -21114.696,E2 -21114.696} C_VEL
LIN {X 0,Y 206.724,Z 369.733,A -85,B 0,C 180,E1 -21119.34,E2 -21119.34} C_VEL
LIN {X 0,Y 206.733,Z 369.73,A -85,B 0,C 180,E1 -21123.773,E2 -21123.773} C_VEL
LIN {X 0,Y 206.759,Z 369.73,A -85,B 0,C 180,E1 -21128.044,E2 -21128.044} C_VEL
LIN {X 0,Y 206.875,Z 369.714,A -85,B 0,C 180,E1 -21132.197,E2 -21132.197} C_VEL
LIN {X 0,Y 206.915,Z 369.709,A -85,B 0,C 180,E1 -21136.246,E2 -21136.246} C_VEL
LIN {X 0,Y 207.134,Z 369.68,A -85,B 0,C 180,E1 -21140.233,E2 -21140.233} C_VEL
LIN {X 0,Y 207.191,Z 369.676,A -85,B 0,C 180,E1 -21142.202,E2 -21142.202} C_VEL
LIN {X 0,Y 207.387,Z 369.651,A -85,B 0,C 180,E1 -21148.058,E2 -21148.058} C_VEL
LIN {X 0,Y 207.521,Z 369.635,A -85,B 0,C 180,E1 -21150,E2 -21150} C_VEL
LIN {X 0,Y 207.088,Z 369.683,A -85,B 0,C 180,E1 -21153.892,E2 -21153.892} C_VEL
LIN {X 0,Y 207.165,Z 369.68,A -85,B 0,C 180,E1 -21157.799,E2 -21157.799} C_VEL
LIN {X 0,Y 206.945,Z 369.703,A -85,B 0,C 180,E1 -21161.757,E2 -21161.757} C_VEL
LIN {X 0,Y 206.869,Z 369.715,A -85,B 0,C 180,E1 -21165.77,E2 -21165.77} C_VEL
LIN {X 0,Y 206.801,Z 369.724,A -85,B 0,C 180,E1 -21169.867,E2 -21169.867} C_VEL
LIN {X 0,Y 206.764,Z 369.728,A -85,B 0,C 180,E1 -21174.071,E2 -21174.071} C_VEL
LIN {X 0,Y 206.737,Z 369.732,A -85,B 0,C 180,E1 -21178.419,E2 -21178.419} C_VEL
LIN {X 0,Y 206.707,Z 369.737,A -85,B 0,C 180,E1 -21182.955,E2 -21182.955} C_VEL
LIN {X 0,Y 206.809,Z 369.98,A -85,B 0,C 180,E1 -21185.168,E2 -21185.168} C_VEL
LIN {X 0,Y 207.132,Z 371.184,A -85,B 0,C 180,E1 -21185.503,E2 -21185.503} C_VEL
LIN {X 0,Y 210.885,Z 383.9,A -85,B 0,C 180,E1 -21187.459,E2 -21187.459} C_VEL
LIN {X 0,Y 213.845,Z 395.119,A -85,B 0,C 180,E1 -21189.507,E2 -21189.507} C_VEL
LIN {X 0,Y 214.388,Z 397.364,A -85,B 0,C 180,E1 -21189.955,E2 -21189.955} C_VEL
LIN {X 0,Y 213.36,Z 405.914,A -85,B 0,C 180,E1 -21191.592,E2 -21191.592} C_VEL
LIN {X 0,Y 211.87,Z 415.663,A -85,B 0,C 180,E1 -21193.8,E2 -21193.8} C_VEL
LIN {X 0,Y 210.322,Z 425.589,A -85,B 0,C 180,E1 -21196.586,E2 -21196.586} C_VEL
LIN {X 0,Y 208.989,Z 434.39,A -85,B 0,C 180,E1 -21199.658,E2 -21199.658} C_VEL
LIN {X 0,Y 208.066,Z 441.006,A -85,B 0,C 180,E1 -21202.555,E2 -21202.555} C_VEL
LIN {X 0,Y 207.393,Z 447.237,A -85,B 0,C 180,E1 -21206.004,E2 -21206.004} C_VEL
LIN {X 0,Y 207.177,Z 451.924,A -85,B 0,C 180,E1 -21209.413,E2 -21209.413} C_VEL
LIN {X 0,Y 207.306,Z 454.375,A -85,B 0,C 180,E1 -21211.814,E2 -21211.814} C_VEL
LIN {X 0,Y 207.626,Z 456.041,A -85,B 0,C 180,E1 -21213.893,E2 -21213.893} C_VEL
LIN {X 0,Y 208.169,Z 457.263,A -85,B 0,C 180,E1 -21216.101,E2 -21216.101} C_VEL
LIN {X 0,Y 209.634,Z 458.236,A -85,B 0,C 180,E1 -21219.831,E2 -21219.831} C_VEL
LIN {X 0,Y 211.112,Z 458.003,A -85,B 0,C 180,E1 -21222.566,E2 -21222.566} C_VEL
LIN {X 0,Y 212.493,Z 457.318,A -85,B 0,C 180,E1 -21224.657,E2 -21224.657} C_VEL
LIN {X 0,Y 215.4,Z 454.935,A -85,B 0,C 180,E1 -21228.183,E2 -21228.183} C_VEL
LIN {X 0,Y 219.065,Z 451.009,A -85,B 0,C 180,E1 -21231.681,E2 -21231.681} C_VEL
LIN {X 0,Y 222.675,Z 446.302,A -85,B 0,C 180,E1 -21234.567,E2 -21234.567} C_VEL
LIN {X 0,Y 226.717,Z 440.255,A -85,B 0,C 180,E1 -21237.335,E2 -21237.335} C_VEL
LIN {X 0,Y 231.186,Z 432.658,A -85,B 0,C 180,E1 -21240,E2 -21240} C_VEL
LIN {X 0,Y 234.15,Z 426.732,A -85,B 0,C 180,E1 -21241.72,E2 -21241.72} C_VEL
LIN {X 0,Y 233.905,Z 418.542,A -85,B 0,C 180,E1 -21245.172,E2 -21245.172} C_VEL
LIN {X 0,Y 232.724,Z 412.845,A -85,B 0,C 180,E1 -21247.848,E2 -21247.848} C_VEL
LIN {X 0,Y 231.283,Z 407.496,A -85,B 0,C 180,E1 -21250.505,E2 -21250.505} C_VEL
LIN {X 0,Y 228.866,Z 401.264,A -85,B 0,C 180,E1 -21254.221,E2 -21254.221} C_VEL
LIN {X 0,Y 227.212,Z 398.517,A -85,B 0,C 180,E1 -21256.494,E2 -21256.494} C_VEL
LIN {X 0,Y 224.568,Z 396.044,A -85,B 0,C 180,E1 -21260.142,E2 -21260.142} C_VEL
LIN {X 0,Y 222.581,Z 394.604,A -85,B 0,C 180,E1 -21264.235,E2 -21264.235} C_VEL
LIN {X 0,Y 221.263,Z 395.682,A -85,B 0,C 180,E1 -21268.454,E2 -21268.454} C_VEL
LIN {X 0,Y 221.154,Z 396.991,A -85,B 0,C 180,E1 -21270.907,E2 -21270.907} C_VEL
LIN {X 0,Y 221.779,Z 400.254,A -85,B 0,C 180,E1 -21274.779,E2 -21274.779} C_VEL
LIN {X 0,Y 223.729,Z 405.079,A -85,B 0,C 180,E1 -21278.922,E2 -21278.922} C_VEL
LIN {X 0,Y 226.348,Z 413.124,A -85,B 0,C 180,E1 -21283.086,E2 -21283.086} C_VEL
LIN {X 0,Y 228.456,Z 420.758,A -85,B 0,C 180,E1 -21286.099,E2 -21286.099} C_VEL
LIN {X 0,Y 228.648,Z 431.379,A -85,B 0,C 180,E1 -21288.809,E2 -21288.809} C_VEL
LIN {X 0,Y 228.086,Z 442.911,A -85,B 0,C 180,E1 -21291.557,E2 -21291.557} C_VEL
LIN {X 0,Y 226.844,Z 452.937,A -85,B 0,C 180,E1 -21293.94,E2 -21293.94} C_VEL
LIN {X 0,Y 224.901,Z 462.585,A -85,B 0,C 180,E1 -21296.313,E2 -21296.313} C_VEL
LIN {X 0,Y 222.063,Z 472.426,A -85,B 0,C 180,E1 -21298.936,E2 -21298.936} C_VEL
LIN {X 0,Y 218.459,Z 481.554,A -85,B 0,C 180,E1 -21301.673,E2 -21301.673} C_VEL
LIN {X 0,Y 214.728,Z 489.911,A -85,B 0,C 180,E1 -21304.748,E2 -21304.748} C_VEL
LIN {X 0,Y 212.511,Z 492.986,A -85,B 0,C 180,E1 -21305.976,E2 -21305.976} C_VEL
LIN {X 0,Y 207.356,Z 497.503,A -85,B 0,C 180,E1 -21307.953,E2 -21307.953} C_VEL
LIN {X 0,Y 202.535,Z 501.281,A -85,B 0,C 180,E1 -21310.117,E2 -21310.117} C_VEL
LIN {X 0,Y 200.879,Z 503.305,A -85,B 0,C 180,E1 -21311.607,E2 -21311.607} C_VEL
LIN {X 0,Y 199.806,Z 505.658,A -85,B 0,C 180,E1 -21313.657,E2 -21313.657} C_VEL
LIN {X 0,Y 198.482,Z 509.069,A -85,B 0,C 180,E1 -21317.734,E2 -21317.734} C_VEL
LIN {X 0,Y 198.39,Z 511.064,A -85,B 0,C 180,E1 -21321.854,E2 -21321.854} C_VEL
LIN {X 0,Y 198.754,Z 511.525,A -85,B 0,C 180,E1 -21323.911,E2 -21323.911} C_VEL
LIN {X 0,Y 199.797,Z 511.211,A -85,B 0,C 180,E1 -21327.984,E2 -21327.984} C_VEL
LIN {X 0,Y 200.431,Z 510.43,A -85,B 0,C 180,E1 -21330,E2 -21330} C_VEL
LIN {X 0,Y 200.021,Z 509.008,A -85,B 0,C 180,E1 -21332.014,E2 -21332.014} C_VEL
LIN {X 0,Y 199.55,Z 505.935,A -85,B 0,C 180,E1 -21335.051,E2 -21335.051} C_VEL
LIN {X 0,Y 199.066,Z 500.699,A -85,B 0,C 180,E1 -21338.682,E2 -21338.682} C_VEL
LIN {X 0,Y 199.264,Z 493.922,A -85,B 0,C 180,E1 -21342.217,E2 -21342.217} C_VEL
LIN {X 0,Y 199.972,Z 486.373,A -85,B 0,C 180,E1 -21345.283,E2 -21345.283} C_VEL
LIN {X 0,Y 201.357,Z 477.009,A -85,B 0,C 180,E1 -21348.308,E2 -21348.308} C_VEL
LIN {X 0,Y 201.873,Z 471.76,A -85,B 0,C 180,E1 -21349.732,E2 -21349.732} C_VEL
LIN {X 0,Y 201.84,Z 462.072,A -85,B 0,C 180,E1 -21351.981,E2 -21351.981} C_VEL
LIN {X 0,Y 201.759,Z 450.705,A -85,B 0,C 180,E1 -21354.16,E2 -21354.16} C_VEL
LIN {X 0,Y 201.519,Z 439.628,A -85,B 0,C 180,E1 -21355.899,E2 -21355.899} C_VEL
LIN {X 0,Y 201.035,Z 426.286,A -85,B 0,C 180,E1 -21357.557,E2 -21357.557} C_VEL
LIN {X 0,Y 200.368,Z 412.236,A -85,B 0,C 180,E1 -21358.871,E2 -21358.871} C_VEL
LIN {X 0,Y 200.112,Z 406.385,A -85,B 0,C 180,E1 -21359.383,E2 -21359.383} C_VEL
LIN {X 0,Y 200.978,Z 401.438,A -85,B 0,C 180,E1 -21362.362,E2 -21362.362} C_VEL
LIN {X 0,Y 203.032,Z 392.932,A -85,B 0,C 180,E1 -21367.731,E2 -21367.731} C_VEL
LIN {X 0,Y 203.54,Z 390.297,A -85,B 0,C 180,E1 -21369.419,E2 -21369.419} C_VEL
LIN {X 0,Y 202.447,Z 384.698,A -85,B 0,C 180,E1 -21373.195,E2 -21373.195} C_VEL
LIN {X 0,Y 200.958,Z 377.363,A -85,B 0,C 180,E1 -21378.358,E2 -21378.358} C_VEL
LIN {X 0,Y 199.724,Z 370.678,A -85,B 0,C 180,E1 -21383.381,E2 -21383.381} C_VEL
LIN {X 0,Y 199.698,Z 370.608,A -85,B 0,C 180,E1 -21388.136,E2 -21388.136} C_VEL
LIN {X 0,Y 199.683,Z 370.61,A -85,B 0,C 180,E1 -21392.771,E2 -21392.771} C_VEL
LIN {X 0,Y 199.708,Z 370.605,A -85,B 0,C 180,E1 -21397.225,E2 -21397.225} C_VEL
LIN {X 0,Y 199.746,Z 370.602,A -85,B 0,C 180,E1 -21401.798,E2 -21401.798} C_VEL
LIN {X 0,Y 199.808,Z 370.589,A -85,B 0,C 180,E1 -21405.746,E2 -21405.746} C_VEL
LIN {X 0,Y 200.019,Z 370.566,A -85,B 0,C 180,E1 -21409.881,E2 -21409.881} C_VEL
LIN {X 0,Y 200.01,Z 370.569,A -85,B 0,C 180,E1 -21413.949,E2 -21413.949} C_VEL
LIN {X 0,Y 200.313,Z 370.529,A -85,B 0,C 180,E1 -21417.989,E2 -21417.989} C_VEL
LIN {X 0,Y 200.474,Z 370.511,A -85,B 0,C 180,E1 -21420,E2 -21420} C_VEL
LIN {X 0,Y 200.021,Z 370.566,A -85,B 0,C 180,E1 -21424.03,E2 -21424.03} C_VEL
LIN {X 0,Y 200.106,Z 370.557,A -85,B 0,C 180,E1 -21428.076,E2 -21428.076} C_VEL
LIN {X 0,Y 199.909,Z 370.582,A -85,B 0,C 180,E1 -21432.177,E2 -21432.177} C_VEL
LIN {X 0,Y 199.799,Z 370.597,A -85,B 0,C 180,E1 -21436.344,E2 -21436.344} C_VEL
LIN {X 0,Y 199.696,Z 370.608,A -85,B 0,C 180,E1 -21440.606,E2 -21440.606} C_VEL
LIN {X 0,Y 199.669,Z 370.612,A -85,B 0,C 180,E1 -21444.985,E2 -21444.985} C_VEL
LIN {X 0,Y 199.672,Z 370.608,A -85,B 0,C 180,E1 -21449.523,E2 -21449.523} C_VEL
LIN {X 0,Y 199.661,Z 370.615,A -85,B 0,C 180,E1 -21452.353,E2 -21452.353} C_VEL
LIN {X 0,Y 199.65,Z 370.613,A -85,B 0,C 180,E1 -21456.757,E2 -21456.757} C_VEL
LIN {X 0,Y 199.672,Z 370.609,A -85,B 0,C 180,E1 -21459.313,E2 -21459.313} C_VEL
LIN {X 0,Y 199.599,Z 370.619,A -85,B 0,C 180,E1 -21464.766,E2 -21464.766} C_VEL
LIN {X 0,Y 199.578,Z 370.623,A -85,B 0,C 180,E1 -21468.006,E2 -21468.006} C_VEL
LIN {X 0,Y 199.639,Z 370.616,A -85,B 0,C 180,E1 -21470.758,E2 -21470.758} C_VEL
LIN {X 0,Y 199.634,Z 370.614,A -85,B 0,C 180,E1 -21475.719,E2 -21475.719} C_VEL
LIN {X 0,Y 199.703,Z 370.61,A -85,B 0,C 180,E1 -21478.138,E2 -21478.138} C_VEL
LIN {X 0,Y 199.687,Z 370.605,A -85,B 0,C 180,E1 -21482.773,E2 -21482.773} C_VEL
LIN {X 0,Y 199.739,Z 370.603,A -85,B 0,C 180,E1 -21487.23,E2 -21487.23} C_VEL
LIN {X 0,Y 199.798,Z 370.595,A -85,B 0,C 180,E1 -21491.758,E2 -21491.758} C_VEL
LIN {X 0,Y 199.85,Z 370.592,A -85,B 0,C 180,E1 -21495.75,E2 -21495.75} C_VEL
LIN {X 0,Y 200.077,Z 370.56,A -85,B 0,C 180,E1 -21499.885,E2 -21499.885} C_VEL
LIN {X 0,Y 200.134,Z 370.556,A -85,B 0,C 180,E1 -21501.925,E2 -21501.925} C_VEL
LIN {X 0,Y 200.327,Z 370.531,A -85,B 0,C 180,E1 -21507.99,E2 -21507.99} C_VEL
LIN {X 0,Y 200.485,Z 370.511,A -85,B 0,C 180,E1 -21510,E2 -21510} C_VEL
LIN {X 0,Y 200.033,Z 370.561,A -85,B 0,C 180,E1 -21514.029,E2 -21514.029} C_VEL
LIN {X 0,Y 200.109,Z 370.558,A -85,B 0,C 180,E1 -21518.076,E2 -21518.076} C_VEL
LIN {X 0,Y 200.037,Z 370.565,A -85,B 0,C 180,E1 -21520.347,E2 -21520.347} C_VEL
LIN {X 0,Y 199.807,Z 370.594,A -85,B 0,C 180,E1 -21526.343,E2 -21526.343} C_VEL
LIN {X 0,Y 199.825,Z 370.593,A -85,B 0,C 180,E1 -21528.453,E2 -21528.453} C_VEL
LIN {X 0,Y 199.737,Z 370.604,A -85,B 0,C 180,E1 -21533.817,E2 -21533.817} C_VEL
LIN {X 0,Y 199.708,Z 370.607,A -85,B 0,C 180,E1 -21538.383,E2 -21538.383} C_VEL
LIN {X 0,Y 199.674,Z 370.614,A -85,B 0,C 180,E1 -21542.356,E2 -21542.356} C_VEL
LIN {X 0,Y 199.738,Z 370.735,A -85,B 0,C 180,E1 -21544.551,E2 -21544.551} C_VEL
LIN {X 0,Y 200.012,Z 371.848,A -85,B 0,C 180,E1 -21544.933,E2 -21544.933} C_VEL
LIN {X 0,Y 203.969,Z 385.271,A -85,B 0,C 180,E1 -21547.083,E2 -21547.083} C_VEL
LIN {X 0,Y 206.955,Z 396.621,A -85,B 0,C 180,E1 -21549.232,E2 -21549.232} C_VEL
LIN {X 0,Y 207.501,Z 399.107,A -85,B 0,C 180,E1 -21549.737,E2 -21549.737} C_VEL
LIN {X 0,Y 205.875,Z 409.842,A -85,B 0,C 180,E1 -21551.929,E2 -21551.929} C_VEL
LIN {X 0,Y 204.293,Z 419.893,A -85,B 0,C 180,E1 -21554.452,E2 -21554.452} C_VEL
LIN {X 0,Y 202.75,Z 429.594,A -85,B 0,C 180,E1 -21557.473,E2 -21557.473} C_VEL
LIN {X 0,Y 201.526,Z 437.564,A -85,B 0,C 180,E1 -21560.565,E2 -21560.565} C_VEL
LIN {X 0,Y 200.764,Z 443.918,A -85,B 0,C 180,E1 -21563.622,E2 -21563.622} C_VEL
LIN {X 0,Y 200.196,Z 450.023,A -85,B 0,C 180,E1 -21567.407,E2 -21567.407} C_VEL
LIN {X 0,Y 200.162,Z 453.856,A -85,B 0,C 180,E1 -21570.557,E2 -21570.557} C_VEL
LIN {X 0,Y 200.38,Z 456.026,A -85,B 0,C 180,E1 -21572.874,E2 -21572.874} C_VEL
LIN {X 0,Y 200.933,Z 457.742,A -85,B 0,C 180,E1 -21575.419,E2 -21575.419} C_VEL
LIN {X 0,Y 201.57,Z 458.708,A -85,B 0,C 180,E1 -21577.448,E2 -21577.448} C_VEL
LIN {X 0,Y 202.514,Z 459.275,A -85,B 0,C 180,E1 -21579.694,E2 -21579.694} C_VEL
LIN {X 0,Y 203.649,Z 459.374,A -85,B 0,C 180,E1 -21581.905,E2 -21581.905} C_VEL
LIN {X 0,Y 205.033,Z 459.003,A -85,B 0,C 180,E1 -21584.084,E2 -21584.084} C_VEL
LIN {X 0,Y 208.248,Z 456.953,A -85,B 0,C 180,E1 -21588.146,E2 -21588.146} C_VEL
LIN {X 0,Y 211.56,Z 453.931,A -85,B 0,C 180,E1 -21591.404,E2 -21591.404} C_VEL
LIN {X 0,Y 215.286,Z 449.783,A -85,B 0,C 180,E1 -21594.38,E2 -21594.38} C_VEL
LIN {X 0,Y 219.502,Z 444.185,A -85,B 0,C 180,E1 -21597.36,E2 -21597.36} C_VEL
LIN {X 0,Y 223.883,Z 437.654,A -85,B 0,C 180,E1 -21600,E2 -21600} C_VEL
LIN {X 0,Y 227.969,Z 430.683,A -85,B 0,C 180,E1 -21602.209,E2 -21602.209} C_VEL
LIN {X 0,Y 228.382,Z 429.432,A -85,B 0,C 180,E1 -21602.646,E2 -21602.646} C_VEL
LIN {X 0,Y 228.591,Z 423.619,A -85,B 0,C 180,E1 -21605.292,E2 -21605.292} C_VEL
LIN {X 0,Y 228.237,Z 419.914,A -85,B 0,C 180,E1 -21607.075,E2 -21607.075} C_VEL
LIN {X 0,Y 226.848,Z 413.082,A -85,B 0,C 180,E1 -21610.713,E2 -21610.713} C_VEL
LIN {X 0,Y 224.989,Z 407.158,A -85,B 0,C 180,E1 -21614.472,E2 -21614.472} C_VEL
LIN {X 0,Y 223.921,Z 404.833,A -85,B 0,C 180,E1 -21616.408,E2 -21616.408} C_VEL
LIN {X 0,Y 221.347,Z 402.342,A -85,B 0,C 180,E1 -21620.442,E2 -21620.442} C_VEL
LIN {X 0,Y 219.617,Z 401.213,A -85,B 0,C 180,E1 -21624.583,E2 -21624.583} C_VEL
LIN {X 0,Y 218.482,Z 402.496,A -85,B 0,C 180,E1 -21628.85,E2 -21628.85} C_VEL
LIN {X 0,Y 218.45,Z 403.715,A -85,B 0,C 180,E1 -21630.981,E2 -21630.981} C_VEL
LIN {X 0,Y 219.14,Z 407.459,A -85,B 0,C 180,E1 -21635.259,E2 -21635.259} C_VEL
LIN {X 0,Y 220.623,Z 411.5,A -85,B 0,C 180,E1 -21638.633,E2 -21638.633} C_VEL
LIN {X 0,Y 222.702,Z 419.171,A -85,B 0,C 180,E1 -21642.728,E2 -21642.728} C_VEL
LIN {X 0,Y 224.013,Z 424.696,A -85,B 0,C 180,E1 -21645.065,E2 -21645.065} C_VEL
LIN {X 0,Y 223.904,Z 432.622,A -85,B 0,C 180,E1 -21647.253,E2 -21647.253} C_VEL
LIN {X 0,Y 222.987,Z 443.477,A -85,B 0,C 180,E1 -21650.059,E2 -21650.059} C_VEL
LIN {X 0,Y 221.256,Z 454.564,A -85,B 0,C 180,E1 -21652.879,E2 -21652.879} C_VEL
LIN {X 0,Y 218.566,Z 465.433,A -85,B 0,C 180,E1 -21655.757,E2 -21655.757} C_VEL
LIN {X 0,Y 215.912,Z 473.359,A -85,B 0,C 180,E1 -21658.032,E2 -21658.032} C_VEL
LIN {X 0,Y 211.603,Z 483.112,A -85,B 0,C 180,E1 -21661.211,E2 -21661.211} C_VEL
LIN {X 0,Y 207.629,Z 491.126,A -85,B 0,C 180,E1 -21664.433,E2 -21664.433} C_VEL
LIN {X 0,Y 203.955,Z 497.569,A -85,B 0,C 180,E1 -21667.726,E2 -21667.726} C_VEL
LIN {X 0,Y 201.554,Z 501.869,A -85,B 0,C 180,E1 -21670.493,E2 -21670.493} C_VEL
LIN {X 0,Y 200.879,Z 503.305,A -85,B 0,C 180,E1 -21671.607,E2 -21671.607} C_VEL
LIN {X 0,Y 199.389,Z 505.128,A -85,B 0,C 180,E1 -21673.158,E2 -21673.158} C_VEL
LIN {X 0,Y 195.477,Z 507.377,A -85,B 0,C 180,E1 -21675.722,E2 -21675.722} C_VEL
LIN {X 0,Y 192.013,Z 508.909,A -85,B 0,C 180,E1 -21678.435,E2 -21678.435} C_VEL
LIN {X 0,Y 191.256,Z 509.551,A -85,B 0,C 180,E1 -21680.175,E2 -21680.175} C_VEL
LIN {X 0,Y 191.689,Z 510.366,A -85,B 0,C 180,E1 -21683.685,E2 -21683.685} C_VEL
LIN {X 0,Y 192.766,Z 509.906,A -85,B 0,C 180,E1 -21687.911,E2 -21687.911} C_VEL
LIN {X 0,Y 193.423,Z 509.077,A -85,B 0,C 180,E1 -21690,E2 -21690} C_VEL
LIN {X 0,Y 192.817,Z 506.606,A -85,B 0,C 180,E1 -21693.134,E2 -21693.134} C_VEL
LIN {X 0,Y 192.331,Z 502.994,A -85,B 0,C 180,E1 -21696.293,E2 -21696.293} C_VEL
LIN {X 0,Y 192.045,Z 497.263,A -85,B 0,C 180,E1 -21699.957,E2 -21699.957} C_VEL
LIN {X 0,Y 192.433,Z 490.72,A -85,B 0,C 180,E1 -21703.194,E2 -21703.194} C_VEL
LIN {X 0,Y 193.291,Z 482.671,A -85,B 0,C 180,E1 -21706.366,E2 -21706.366} C_VEL
LIN {X 0,Y 194.733,Z 473.143,A -85,B 0,C 180,E1 -21709.336,E2 -21709.336} C_VEL
LIN {X 0,Y 194.8,Z 463.82,A -85,B 0,C 180,E1 -21711.703,E2 -21711.703} C_VEL
LIN {X 0,Y 194.73,Z 453.164,A -85,B 0,C 180,E1 -21713.955,E2 -21713.955} C_VEL
LIN {X 0,Y 194.533,Z 441.368,A -85,B 0,C 180,E1 -21715.979,E2 -21715.979} C_VEL
LIN {X 0,Y 194.166,Z 428.27,A -85,B 0,C 180,E1 -21717.775,E2 -21717.775} C_VEL
LIN {X 0,Y 193.547,Z 414.247,A -85,B 0,C 180,E1 -21719.227,E2 -21719.227} C_VEL
LIN {X 0,Y 193.169,Z 405.494,A -85,B 0,C 180,E1 -21719.989,E2 -21719.989} C_VEL
LIN {X 0,Y 193.696,Z 402.568,A -85,B 0,C 180,E1 -21721.742,E2 -21721.742} C_VEL
LIN {X 0,Y 195.382,Z 395.471,A -85,B 0,C 180,E1 -21726.406,E2 -21726.406} C_VEL
LIN {X 0,Y 196.322,Z 391.733,A -85,B 0,C 180,E1 -21728.874,E2 -21728.874} C_VEL
LIN {X 0,Y 196.032,Z 388.367,A -85,B 0,C 180,E1 -21731.159,E2 -21731.159} C_VEL
LIN {X 0,Y 194.807,Z 382.666,A -85,B 0,C 180,E1 -21735.216,E2 -21735.216} C_VEL
LIN {X 0,Y 193.356,Z 375.275,A -85,B 0,C 180,E1 -21740.727,E2 -21740.727} C_VEL
LIN {X 0,Y 192.659,Z 371.531,A -85,B 0,C 180,E1 -21743.812,E2 -21743.812} C_VEL
LIN {X 0,Y 192.603,Z 371.494,A -85,B 0,C 180,E1 -21749.279,E2 -21749.279} C_VEL
LIN {X 0,Y 192.662,Z 371.484,A -85,B 0,C 180,E1 -21751.691,E2 -21751.691} C_VEL
LIN {X 0,Y 192.681,Z 371.481,A -85,B 0,C 180,E1 -21756.345,E2 -21756.345} C_VEL
LIN {X 0,Y 192.694,Z 371.482,A -85,B 0,C 180,E1 -21761.487,E2 -21761.487} C_VEL
LIN {X 0,Y 192.734,Z 371.472,A -85,B 0,C 180,E1 -21765.211,E2 -21765.211} C_VEL
LIN {X 0,Y 192.941,Z 371.448,A -85,B 0,C 180,E1 -21769.566,E2 -21769.566} C_VEL
LIN {X 0,Y 192.972,Z 371.446,A -85,B 0,C 180,E1 -21773.727,E2 -21773.727} C_VEL
LIN {X 0,Y 193.255,Z 371.408,A -85,B 0,C 180,E1 -21777.916,E2 -21777.916} C_VEL
LIN {X 0,Y 193.438,Z 371.388,A -85,B 0,C 180,E1 -21780,E2 -21780} C_VEL
LIN {X 0,Y 192.968,Z 371.445,A -85,B 0,C 180,E1 -21784.177,E2 -21784.177} C_VEL
LIN {X 0,Y 193.056,Z 371.436,A -85,B 0,C 180,E1 -21788.373,E2 -21788.373} C_VEL
LIN {X 0,Y 192.848,Z 371.46,A -85,B 0,C 180,E1 -21792.63,E2 -21792.63} C_VEL
LIN {X 0,Y 192.728,Z 371.479,A -85,B 0,C 180,E1 -21798.543,E2 -21798.543} C_VEL
LIN {X 0,Y 192.661,Z 371.485,A -85,B 0,C 180,E1 -21804.225,E2 -21804.225} C_VEL
LIN {X 0,Y 192.647,Z 371.484,A -85,B 0,C 180,E1 -21808.893,E2 -21808.893} C_VEL
LIN {X 0,Y 192.598,Z 371.493,A -85,B 0,C 180,E1 -21813.186,E2 -21813.186} C_VEL
LIN {X 0,Y 192.596,Z 371.492,A -85,B 0,C 180,E1 -21818.341,E2 -21818.341} C_VEL
LIN {X 0,Y 192.534,Z 371.5,A -85,B 0,C 180,E1 -21823.111,E2 -21823.111} C_VEL
LIN {X 0,Y 192.514,Z 371.5,A -85,B 0,C 180,E1 -21826.897,E2 -21826.897} C_VEL
LIN {X 0,Y 192.572,Z 371.497,A -85,B 0,C 180,E1 -21831.654,E2 -21831.654} C_VEL
LIN {X 0,Y 192.597,Z 371.491,A -85,B 0,C 180,E1 -21834.279,E2 -21834.279} C_VEL
LIN {X 0,Y 192.607,Z 371.492,A -85,B 0,C 180,E1 -21839.281,E2 -21839.281} C_VEL
LIN {X 0,Y 192.665,Z 371.485,A -85,B 0,C 180,E1 -21841.693,E2 -21841.693} C_VEL
LIN {X 0,Y 192.707,Z 371.48,A -85,B 0,C 180,E1 -21846.349,E2 -21846.349} C_VEL
LIN {X 0,Y 192.733,Z 371.474,A -85,B 0,C 180,E1 -21851.458,E2 -21851.458} C_VEL
LIN {X 0,Y 192.774,Z 371.471,A -85,B 0,C 180,E1 -21855.215,E2 -21855.215} C_VEL
LIN {X 0,Y 193.022,Z 371.438,A -85,B 0,C 180,E1 -21859.511,E2 -21859.511} C_VEL
LIN {X 0,Y 193.007,Z 371.445,A -85,B 0,C 180,E1 -21863.729,E2 -21863.729} C_VEL
LIN {X 0,Y 193.269,Z 371.41,A -85,B 0,C 180,E1 -21867.916,E2 -21867.916} C_VEL
LIN {X 0,Y 193.449,Z 371.388,A -85,B 0,C 180,E1 -21870,E2 -21870} C_VEL
LIN {X 0,Y 192.979,Z 371.439,A -85,B 0,C 180,E1 -21874.177,E2 -21874.177} C_VEL
LIN {X 0,Y 193.061,Z 371.435,A -85,B 0,C 180,E1 -21878.373,E2 -21878.373} C_VEL
LIN {X 0,Y 192.811,Z 371.462,A -85,B 0,C 180,E1 -21882.632,E2 -21882.632} C_VEL
LIN {X 0,Y 192.772,Z 371.471,A -85,B 0,C 180,E1 -21886.957,E2 -21886.957} C_VEL
LIN {X 0,Y 192.643,Z 371.489,A -85,B 0,C 180,E1 -21891.396,E2 -21891.396} C_VEL
LIN {X 0,Y 192.665,Z 371.485,A -85,B 0,C 180,E1 -21894.224,E2 -21894.224} C_VEL
LIN {X 0,Y 192.644,Z 371.489,A -85,B 0,C 180,E1 -21898.888,E2 -21898.888} C_VEL
LIN {X 0,Y 192.657,Z 371.59,A -85,B 0,C 180,E1 -21903.957,E2 -21903.957} C_VEL
LIN {X 0,Y 192.943,Z 372.696,A -85,B 0,C 180,E1 -21904.373,E2 -21904.373} C_VEL
LIN {X 0,Y 196.797,Z 385.867,A -85,B 0,C 180,E1 -21906.558,E2 -21906.558} C_VEL
LIN {X 0,Y 199.696,Z 396.738,A -85,B 0,C 180,E1 -21908.675,E2 -21908.675} C_VEL
LIN {X 0,Y 200.465,Z 400.797,A -85,B 0,C 180,E1 -21909.53,E2 -21909.53} C_VEL
LIN {X 0,Y 198.603,Z 412.291,A -85,B 0,C 180,E1 -21912.001,E2 -21912.001} C_VEL
LIN {X 0,Y 197.08,Z 421.736,A -85,B 0,C 180,E1 -21914.503,E2 -21914.503} C_VEL
LIN {X 0,Y 195.564,Z 431.174,A -85,B 0,C 180,E1 -21917.6,E2 -21917.6} C_VEL
LIN {X 0,Y 194.36,Z 438.934,A -85,B 0,C 180,E1 -21920.743,E2 -21920.743} C_VEL
LIN {X 0,Y 193.643,Z 444.822,A -85,B 0,C 180,E1 -21923.684,E2 -21923.684} C_VEL
LIN {X 0,Y 193.153,Z 450.036,A -85,B 0,C 180,E1 -21926.922,E2 -21926.922} C_VEL
LIN {X 0,Y 193.129,Z 454.799,A -85,B 0,C 180,E1 -21930.85,E2 -21930.85} C_VEL
LIN {X 0,Y 193.787,Z 458.305,A -85,B 0,C 180,E1 -21935.045,E2 -21935.045} C_VEL
LIN {X 0,Y 195.279,Z 460.194,A -85,B 0,C 180,E1 -21939.342,E2 -21939.342} C_VEL
LIN {X 0,Y 197.522,Z 460.479,A -85,B 0,C 180,E1 -21943.462,E2 -21943.462} C_VEL
LIN {X 0,Y 199.071,Z 459.952,A -85,B 0,C 180,E1 -21945.692,E2 -21945.692} C_VEL
LIN {X 0,Y 201.088,Z 458.858,A -85,B 0,C 180,E1 -21948.117,E2 -21948.117} C_VEL
LIN {X 0,Y 202.911,Z 457.51,A -85,B 0,C 180,E1 -21950.027,E2 -21950.027} C_VEL
LIN {X 0,Y 206.619,Z 454.175,A -85,B 0,C 180,E1 -21953.317,E2 -21953.317} C_VEL
LIN {X 0,Y 211.188,Z 449.221,A -85,B 0,C 180,E1 -21956.684,E2 -21956.684} C_VEL
LIN {X 0,Y 215.707,Z 443.395,A -85,B 0,C 180,E1 -21959.533,E2 -21959.533} C_VEL
LIN {X 0,Y 220.688,Z 436.007,A -85,B 0,C 180,E1 -21962.281,E2 -21962.281} C_VEL
LIN {X 0,Y 222.441,Z 433.162,A -85,B 0,C 180,E1 -21963.17,E2 -21963.17} C_VEL
LIN {X 0,Y 223.121,Z 428.463,A -85,B 0,C 180,E1 -21965.422,E2 -21965.422} C_VEL
LIN {X 0,Y 222.965,Z 423.832,A -85,B 0,C 180,E1 -21967.847,E2 -21967.847} C_VEL
LIN {X 0,Y 222.118,Z 417.975,A -85,B 0,C 180,E1 -21971.234,E2 -21971.234} C_VEL
LIN {X 0,Y 220.859,Z 412.889,A -85,B 0,C 180,E1 -21974.748,E2 -21974.748} C_VEL
LIN {X 0,Y 220.05,Z 410.711,A -85,B 0,C 180,E1 -21976.705,E2 -21976.705} C_VEL
LIN {X 0,Y 217.842,Z 408.482,A -85,B 0,C 180,E1 -21980.786,E2 -21980.786} C_VEL
LIN {X 0,Y 216.335,Z 407.674,A -85,B 0,C 180,E1 -21984.982,E2 -21984.982} C_VEL
LIN {X 0,Y 215.464,Z 409.212,A -85,B 0,C 180,E1 -21989.293,E2 -21989.293} C_VEL
LIN {X 0,Y 215.433,Z 411.017,A -85,B 0,C 180,E1 -21991.987,E2 -21991.987} C_VEL
LIN {X 0,Y 216.667,Z 415.9,A -85,B 0,C 180,E1 -21996.98,E2 -21996.98} C_VEL
LIN {X 0,Y 217.055,Z 417.146,A -85,B 0,C 180,E1 -21997.967,E2 -21997.967} C_VEL
LIN {X 0,Y 218.753,Z 425.184,A -85,B 0,C 180,E1 -22002.429,E2 -22002.429} C_VEL
LIN {X 0,Y 219.447,Z 429.098,A -85,B 0,C 180,E1 -22004.131,E2 -22004.131} C_VEL
LIN {X 0,Y 219.369,Z 432.379,A -85,B 0,C 180,E1 -22005.186,E2 -22005.186} C_VEL
LIN {X 0,Y 218.425,Z 441.438,A -85,B 0,C 180,E1 -22007.735,E2 -22007.735} C_VEL
LIN {X 0,Y 216.479,Z 452.798,A -85,B 0,C 180,E1 -22010.844,E2 -22010.844} C_VEL
LIN {X 0,Y 213.807,Z 463.157,A -85,B 0,C 180,E1 -22013.725,E2 -22013.725} C_VEL
LIN {X 0,Y 210.42,Z 472.785,A -85,B 0,C 180,E1 -22016.616,E2 -22016.616} C_VEL
LIN {X 0,Y 206.018,Z 482.151,A -85,B 0,C 180,E1 -22019.791,E2 -22019.791} C_VEL
LIN {X 0,Y 201.838,Z 490.051,A -85,B 0,C 180,E1 -22023.086,E2 -22023.086} C_VEL
LIN {X 0,Y 198.369,Z 495.648,A -85,B 0,C 180,E1 -22025.957,E2 -22025.957} C_VEL
LIN {X 0,Y 194.933,Z 501.118,A -85,B 0,C 180,E1 -22029.619,E2 -22029.619} C_VEL
LIN {X 0,Y 192.926,Z 504.947,A -85,B 0,C 180,E1 -22033.057,E2 -22033.057} C_VEL
LIN {X 0,Y 191.491,Z 508.192,A -85,B 0,C 180,E1 -22037.279,E2 -22037.279} C_VEL
LIN {X 0,Y 191.256,Z 509.551,A -85,B 0,C 180,E1 -22040.175,E2 -22040.175} C_VEL
LIN {X 0,Y 190.704,Z 510.006,A -85,B 0,C 180,E1 -22041.935,E2 -22041.935} C_VEL
LIN {X 0,Y 188.358,Z 509.796,A -85,B 0,C 180,E1 -22044.844,E2 -22044.844} C_VEL
LIN {X 0,Y 186.59,Z 508.964,A -85,B 0,C 180,E1 -22047.218,E2 -22047.218} C_VEL
LIN {X 0,Y 186.16,Z 508.133,A -85,B 0,C 180,E1 -22049.032,E2 -22049.032} C_VEL
LIN {X 0,Y 186.297,Z 507.825,A -85,B 0,C 180,E1 -22049.637,E2 -22049.637} C_VEL
LIN {X 0,Y 186.433,Z 507.668,A -85,B 0,C 180,E1 -22050,E2 -22050} C_VEL
LIN {X 0,Y 185.81,Z 505.049,A -85,B 0,C 180,E1 -22053.252,E2 -22053.252} C_VEL
LIN {X 0,Y 185.291,Z 501.252,A -85,B 0,C 180,E1 -22056.534,E2 -22056.534} C_VEL
LIN {X 0,Y 185.069,Z 495.32,A -85,B 0,C 180,E1 -22060.336,E2 -22060.336} C_VEL
LIN {X 0,Y 185.449,Z 488.582,A -85,B 0,C 180,E1 -22063.701,E2 -22063.701} C_VEL
LIN {X 0,Y 186.506,Z 480.271,A -85,B 0,C 180,E1 -22066.98,E2 -22066.98} C_VEL
LIN {X 0,Y 187.576,Z 473.668,A -85,B 0,C 180,E1 -22069.137,E2 -22069.137} C_VEL
LIN {X 0,Y 187.721,Z 464.642,A -85,B 0,C 180,E1 -22071.59,E2 -22071.59} C_VEL
LIN {X 0,Y 187.652,Z 453.79,A -85,B 0,C 180,E1 -22074.034,E2 -22074.034} C_VEL
LIN {X 0,Y 187.511,Z 441.968,A -85,B 0,C 180,E1 -22076.212,E2 -22076.212} C_VEL
LIN {X 0,Y 187.196,Z 428.691,A -85,B 0,C 180,E1 -22078.14,E2 -22078.14} C_VEL
LIN {X 0,Y 186.68,Z 415.459,A -85,B 0,C 180,E1 -22079.625,E2 -22079.625} C_VEL
LIN {X 0,Y 186.227,Z 404.504,A -85,B 0,C 180,E1 -22080.64,E2 -22080.64} C_VEL
LIN {X 0,Y 187.52,Z 398.688,A -85,B 0,C 180,E1 -22084.459,E2 -22084.459} C_VEL
LIN {X 0,Y 189.233,Z 391.833,A -85,B 0,C 180,E1 -22089.15,E2 -22089.15} C_VEL
LIN {X 0,Y 188.763,Z 388.048,A -85,B 0,C 180,E1 -22091.872,E2 -22091.872} C_VEL
LIN {X 0,Y 187.411,Z 381.931,A -85,B 0,C 180,E1 -22096.401,E2 -22096.401} C_VEL
LIN {X 0,Y 186.161,Z 375.451,A -85,B 0,C 180,E1 -22101.471,E2 -22101.471} C_VEL
LIN {X 0,Y 185.611,Z 372.417,A -85,B 0,C 180,E1 -22104.063,E2 -22104.063} C_VEL
LIN {X 0,Y 185.541,Z 372.372,A -85,B 0,C 180,E1 -22107.974,E2 -22107.974} C_VEL
LIN {X 0,Y 185.579,Z 372.366,A -85,B 0,C 180,E1 -22110.575,E2 -22110.575} C_VEL
LIN {X 0,Y 185.577,Z 372.367,A -85,B 0,C 180,E1 -22115.381,E2 -22115.381} C_VEL
LIN {X 0,Y 185.58,Z 372.366,A -85,B 0,C 180,E1 -22120.072,E2 -22120.072} C_VEL
LIN {X 0,Y 185.664,Z 372.356,A -85,B 0,C 180,E1 -22124.634,E2 -22124.634} C_VEL
LIN {X 0,Y 185.884,Z 372.328,A -85,B 0,C 180,E1 -22129.419,E2 -22129.419} C_VEL
LIN {X 0,Y 185.935,Z 372.323,A -85,B 0,C 180,E1 -22133.489,E2 -22133.489} C_VEL
LIN {X 0,Y 186.198,Z 372.287,A -85,B 0,C 180,E1 -22137.837,E2 -22137.837} C_VEL
LIN {X 0,Y 186.401,Z 372.264,A -85,B 0,C 180,E1 -22140,E2 -22140} C_VEL
LIN {X 0,Y 185.915,Z 372.324,A -85,B 0,C 180,E1 -22144.336,E2 -22144.336} C_VEL
LIN {X 0,Y 186.004,Z 372.317,A -85,B 0,C 180,E1 -22148.693,E2 -22148.693} C_VEL
LIN {X 0,Y 185.759,Z 372.341,A -85,B 0,C 180,E1 -22153.121,E2 -22153.121} C_VEL
LIN {X 0,Y 185.671,Z 372.356,A -85,B 0,C 180,E1 -22158.867,E2 -22158.867} C_VEL
LIN {X 0,Y 185.598,Z 372.367,A -85,B 0,C 180,E1 -22164.663,E2 -22164.663} C_VEL
LIN {X 0,Y 185.576,Z 372.364,A -85,B 0,C 180,E1 -22169.494,E2 -22169.494} C_VEL
LIN {X 0,Y 185.518,Z 372.376,A -85,B 0,C 180,E1 -22174.628,E2 -22174.628} C_VEL
LIN {X 0,Y 185.542,Z 372.369,A -85,B 0,C 180,E1 -22177.305,E2 -22177.305} C_VEL
LIN {X 0,Y 185.51,Z 372.376,A -85,B 0,C 180,E1 -22180.74,E2 -22180.74} C_VEL
LIN {X 0,Y 185.485,Z 372.377,A -85,B 0,C 180,E1 -22186.047,E2 -22186.047} C_VEL
LIN {X 0,Y 185.487,Z 372.38,A -85,B 0,C 180,E1 -22189.901,E2 -22189.901} C_VEL
LIN {X 0,Y 185.543,Z 372.37,A -85,B 0,C 180,E1 -22192.697,E2 -22192.697} C_VEL
LIN {X 0,Y 185.545,Z 372.374,A -85,B 0,C 180,E1 -22197.976,E2 -22197.976} C_VEL
LIN {X 0,Y 185.582,Z 372.366,A -85,B 0,C 180,E1 -22200.576,E2 -22200.576} C_VEL
LIN {X 0,Y 185.588,Z 372.365,A -85,B 0,C 180,E1 -22205.383,E2 -22205.383} C_VEL
LIN {X 0,Y 185.676,Z 372.351,A -85,B 0,C 180,E1 -22211.133,E2 -22211.133} C_VEL
LIN {X 0,Y 185.726,Z 372.349,A -85,B 0,C 180,E1 -22214.64,E2 -22214.64} C_VEL
LIN {X 0,Y 185.944,Z 372.32,A -85,B 0,C 180,E1 -22219.329,E2 -22219.329} C_VEL
LIN {X 0,Y 185.972,Z 372.321,A -85,B 0,C 180,E1 -22223.49,E2 -22223.49} C_VEL
LIN {X 0,Y 186.213,Z 372.289,A -85,B 0,C 180,E1 -22227.837,E2 -22227.837} C_VEL
LIN {X 0,Y 186.412,Z 372.265,A -85,B 0,C 180,E1 -22230,E2 -22230} C_VEL
LIN {X 0,Y 185.926,Z 372.317,A -85,B 0,C 180,E1 -22234.336,E2 -22234.336} C_VEL
LIN {X 0,Y 186.008,Z 372.314,A -85,B 0,C 180,E1 -22238.692,E2 -22238.692} C_VEL
LIN {X 0,Y 185.736,Z 372.345,A -85,B 0,C 180,E1 -22243.122,E2 -22243.122} C_VEL
LIN {X 0,Y 185.718,Z 372.351,A -85,B 0,C 180,E1 -22247.622,E2 -22247.622} C_VEL
LIN {X 0,Y 185.601,Z 372.365,A -85,B 0,C 180,E1 -22252.25,E2 -22252.25} C_VEL
LIN {X 0,Y 185.561,Z 372.372,A -85,B 0,C 180,E1 -22257.032,E2 -22257.032} C_VEL
LIN {X 0,Y 185.577,Z 372.369,A -85,B 0,C 180,E1 -22259.493,E2 -22259.493} C_VEL
LIN {X 0,Y 185.61,Z 372.496,A -85,B 0,C 180,E1 -22263.388,E2 -22263.388} C_VEL
LIN {X 0,Y 185.893,Z 373.682,A -85,B 0,C 180,E1 -22263.808,E2 -22263.808} C_VEL
LIN {X 0,Y 189.713,Z 386.599,A -85,B 0,C 180,E1 -22266.021,E2 -22266.021} C_VEL
LIN {X 0,Y 192.728,Z 397.885,A -85,B 0,C 180,E1 -22268.309,E2 -22268.309} C_VEL
LIN {X 0,Y 193.52,Z 401.619,A -85,B 0,C 180,E1 -22269.132,E2 -22269.132} C_VEL
LIN {X 0,Y 191.703,Z 412.585,A -85,B 0,C 180,E1 -22271.55,E2 -22271.55} C_VEL
LIN {X 0,Y 189.995,Z 422.908,A -85,B 0,C 180,E1 -22274.362,E2 -22274.362} C_VEL
LIN {X 0,Y 188.627,Z 431.207,A -85,B 0,C 180,E1 -22277.159,E2 -22277.159} C_VEL
LIN {X 0,Y 187.356,Z 439.024,A -85,B 0,C 180,E1 -22280.38,E2 -22280.38} C_VEL
LIN {X 0,Y 186.566,Z 445.379,A -85,B 0,C 180,E1 -22283.608,E2 -22283.608} C_VEL
LIN {X 0,Y 186.075,Z 450.919,A -85,B 0,C 180,E1 -22287.112,E2 -22287.112} C_VEL
LIN {X 0,Y 186.039,Z 455.173,A -85,B 0,C 180,E1 -22290.587,E2 -22290.587} C_VEL
LIN {X 0,Y 186.617,Z 458.735,A -85,B 0,C 180,E1 -22294.664,E2 -22294.664} C_VEL
LIN {X 0,Y 188.081,Z 461.057,A -85,B 0,C 180,E1 -22299.091,E2 -22299.091} C_VEL
LIN {X 0,Y 190.488,Z 461.703,A -85,B 0,C 180,E1 -22303.584,E2 -22303.584} C_VEL
LIN {X 0,Y 193.32,Z 460.911,A -85,B 0,C 180,E1 -22307.401,E2 -22307.401} C_VEL
LIN {X 0,Y 195.336,Z 459.78,A -85,B 0,C 180,E1 -22309.636,E2 -22309.636} C_VEL
LIN {X 0,Y 198.452,Z 457.552,A -85,B 0,C 180,E1 -22312.554,E2 -22312.554} C_VEL
LIN {X 0,Y 202.992,Z 453.467,A -85,B 0,C 180,E1 -22316.029,E2 -22316.029} C_VEL
LIN {X 0,Y 207.479,Z 448.538,A -85,B 0,C 180,E1 -22319.03,E2 -22319.03} C_VEL
LIN {X 0,Y 212.531,Z 442.207,A -85,B 0,C 180,E1 -22321.895,E2 -22321.895} C_VEL
LIN {X 0,Y 216.974,Z 435.751,A -85,B 0,C 180,E1 -22324.179,E2 -22324.179} C_VEL
LIN {X 0,Y 217.66,Z 431.391,A -85,B 0,C 180,E1 -22326.489,E2 -22326.489} C_VEL
LIN {X 0,Y 217.634,Z 426.695,A -85,B 0,C 180,E1 -22329.292,E2 -22329.292} C_VEL
LIN {X 0,Y 217.27,Z 422.283,A -85,B 0,C 180,E1 -22332.137,E2 -22332.137} C_VEL
LIN {X 0,Y 216.349,Z 417.508,A -85,B 0,C 180,E1 -22335.87,E2 -22335.87} C_VEL
LIN {X 0,Y 215.936,Z 416.417,A -85,B 0,C 180,E1 -22337.033,E2 -22337.033} C_VEL
LIN {X 0,Y 214.04,Z 414.487,A -85,B 0,C 180,E1 -22341.173,E2 -22341.173} C_VEL
LIN {X 0,Y 213.371,Z 414.046,A -85,B 0,C 180,E1 -22343.282,E2 -22343.282} C_VEL
LIN {X 0,Y 212.778,Z 414.055,A -85,B 0,C 180,E1 -22345.429,E2 -22345.429} C_VEL
LIN {X 0,Y 212.083,Z 415.884,A -85,B 0,C 180,E1 -22349.806,E2 -22349.806} C_VEL
LIN {X 0,Y 212.058,Z 417.422,A -85,B 0,C 180,E1 -22352.024,E2 -22352.024} C_VEL
LIN {X 0,Y 212.937,Z 421.645,A -85,B 0,C 180,E1 -22356.448,E2 -22356.448} C_VEL
LIN {X 0,Y 213.327,Z 423.341,A -85,B 0,C 180,E1 -22357.753,E2 -22357.753} C_VEL
LIN {X 0,Y 214.422,Z 430.047,A -85,B 0,C 180,E1 -22361.653,E2 -22361.653} C_VEL
LIN {X 0,Y 214.868,Z 433.737,A -85,B 0,C 180,E1 -22363.384,E2 -22363.384} C_VEL
LIN {X 0,Y 214.388,Z 438.331,A -85,B 0,C 180,E1 -22364.882,E2 -22364.882} C_VEL
LIN {X 0,Y 212.449,Z 448.911,A -85,B 0,C 180,E1 -22368.015,E2 -22368.015} C_VEL
LIN {X 0,Y 210.273,Z 457.626,A -85,B 0,C 180,E1 -22370.578,E2 -22370.578} C_VEL
LIN {X 0,Y 207.002,Z 467.461,A -85,B 0,C 180,E1 -22373.549,E2 -22373.549} C_VEL
LIN {X 0,Y 203.285,Z 476.089,A -85,B 0,C 180,E1 -22376.417,E2 -22376.417} C_VEL
LIN {X 0,Y 198.597,Z 484.79,A -85,B 0,C 180,E1 -22379.717,E2 -22379.717} C_VEL
LIN {X 0,Y 194.235,Z 491.916,A -85,B 0,C 180,E1 -22383.11,E2 -22383.11} C_VEL
LIN {X 0,Y 189.816,Z 498.395,A -85,B 0,C 180,E1 -22387.123,E2 -22387.123} C_VEL
LIN {X 0,Y 187.298,Z 502.186,A -85,B 0,C 180,E1 -22390.263,E2 -22390.263} C_VEL
LIN {X 0,Y 185.133,Z 505.961,A -85,B 0,C 180,E1 -22394.59,E2 -22394.59} C_VEL
LIN {X 0,Y 184.251,Z 508.285,A -85,B 0,C 180,E1 -22399.006,E2 -22399.006} C_VEL
LIN {X 0,Y 184.626,Z 509.193,A -85,B 0,C 180,E1 -22403.443,E2 -22403.443} C_VEL
LIN {X 0,Y 185.731,Z 508.605,A -85,B 0,C 180,E1 -22407.831,E2 -22407.831} C_VEL
LIN {X 0,Y 186.297,Z 507.825,A -85,B 0,C 180,E1 -22409.637,E2 -22409.637} C_VEL
LIN {X 0,Y 186.254,Z 507.124,A -85,B 0,C 180,E1 -22410.812,E2 -22410.812} C_VEL
LIN {X 0,Y 185.48,Z 506.129,A -85,B 0,C 180,E1 -22411.951,E2 -22411.951} C_VEL
LIN {X 0,Y 182.713,Z 503.541,A -85,B 0,C 180,E1 -22414.127,E2 -22414.127} C_VEL
LIN {X 0,Y 179.625,Z 500.368,A -85,B 0,C 180,E1 -22416.322,E2 -22416.322} C_VEL
LIN {X 0,Y 178.219,Z 497.742,A -85,B 0,C 180,E1 -22418.036,E2 -22418.036} C_VEL
LIN {X 0,Y 178.082,Z 496.833,A -85,B 0,C 180,E1 -22418.624,E2 -22418.624} C_VEL
LIN {X 0,Y 178.208,Z 491.106,A -85,B 0,C 180,E1 -22421.949,E2 -22421.949} C_VEL
LIN {X 0,Y 178.86,Z 483.683,A -85,B 0,C 180,E1 -22425.38,E2 -22425.38} C_VEL
LIN {X 0,Y 180.285,Z 474.451,A -85,B 0,C 180,E1 -22428.76,E2 -22428.76} C_VEL
LIN {X 0,Y 180.643,Z 468.775,A -85,B 0,C 180,E1 -22430.496,E2 -22430.496} C_VEL
LIN {X 0,Y 180.598,Z 458.284,A -85,B 0,C 180,E1 -22433.204,E2 -22433.204} C_VEL
LIN {X 0,Y 180.587,Z 446.505,A -85,B 0,C 180,E1 -22435.698,E2 -22435.698} C_VEL
LIN {X 0,Y 180.341,Z 433.542,A -85,B 0,C 180,E1 -22437.881,E2 -22437.881} C_VEL
LIN {X 0,Y 179.981,Z 421.105,A -85,B 0,C 180,E1 -22439.536,E2 -22439.536} C_VEL
LIN {X 0,Y 179.413,Z 407.009,A -85,B 0,C 180,E1 -22440.939,E2 -22440.939} C_VEL
LIN {X 0,Y 179.297,Z 403.627,A -85,B 0,C 180,E1 -22441.289,E2 -22441.289} C_VEL
LIN {X 0,Y 179.874,Z 400.73,A -85,B 0,C 180,E1 -22443.161,E2 -22443.161} C_VEL
LIN {X 0,Y 181.786,Z 393.672,A -85,B 0,C 180,E1 -22448.211,E2 -22448.211} C_VEL
LIN {X 0,Y 182.072,Z 390.956,A -85,B 0,C 180,E1 -22450.17,E2 -22450.17} C_VEL
LIN {X 0,Y 181.176,Z 386.428,A -85,B 0,C 180,E1 -22453.587,E2 -22453.587} C_VEL
LIN {X 0,Y 179.856,Z 380.332,A -85,B 0,C 180,E1 -22458.372,E2 -22458.372} C_VEL
LIN {X 0,Y 178.953,Z 375.306,A -85,B 0,C 180,E1 -22462.502,E2 -22462.502} C_VEL
LIN {X 0,Y 178.55,Z 373.295,A -85,B 0,C 180,E1 -22464.36,E2 -22464.36} C_VEL
LIN {X 0,Y 178.52,Z 373.245,A -85,B 0,C 180,E1 -22470.006,E2 -22470.006} C_VEL
LIN {X 0,Y 178.517,Z 373.249,A -85,B 0,C 180,E1 -22474.885,E2 -22474.885} C_VEL
LIN {X 0,Y 178.587,Z 373.239,A -85,B 0,C 180,E1 -22480.814,E2 -22480.814} C_VEL
LIN {X 0,Y 178.639,Z 373.225,A -85,B 0,C 180,E1 -22486.346,E2 -22486.346} C_VEL
LIN {X 0,Y 178.901,Z 373.2,A -85,B 0,C 180,E1 -22490.959,E2 -22490.959} C_VEL
LIN {X 0,Y 179.144,Z 373.166,A -85,B 0,C 180,E1 -22497.752,E2 -22497.752} C_VEL
LIN {X 0,Y 179.364,Z 373.141,A -85,B 0,C 180,E1 -22500,E2 -22500} C_VEL
LIN {X 0,Y 178.864,Z 373.202,A -85,B 0,C 180,E1 -22504.507,E2 -22504.507} C_VEL
LIN {X 0,Y 178.933,Z 373.196,A -85,B 0,C 180,E1 -22509.039,E2 -22509.039} C_VEL
LIN {X 0,Y 178.676,Z 373.222,A -85,B 0,C 180,E1 -22513.651,E2 -22513.651} C_VEL
LIN {X 0,Y 178.62,Z 373.233,A -85,B 0,C 180,E1 -22519.216,E2 -22519.216} C_VEL
LIN {X 0,Y 178.532,Z 373.245,A -85,B 0,C 180,E1 -22525.125,E2 -22525.125} C_VEL
LIN {X 0,Y 178.476,Z 373.251,A -85,B 0,C 180,E1 -22530.791,E2 -22530.791} C_VEL
LIN {X 0,Y 178.495,Z 373.252,A -85,B 0,C 180,E1 -22534.226,E2 -22534.226} C_VEL
LIN {X 0,Y 178.435,Z 373.254,A -85,B 0,C 180,E1 -22539.064,E2 -22539.064} C_VEL
LIN {X 0,Y 178.427,Z 373.26,A -85,B 0,C 180,E1 -22542.037,E2 -22542.037} C_VEL
LIN {X 0,Y 178.416,Z 373.257,A -85,B 0,C 180,E1 -22545.157,E2 -22545.157} C_VEL
LIN {X 0,Y 178.413,Z 373.261,A -85,B 0,C 180,E1 -22548.456,E2 -22548.456} C_VEL
LIN {X 0,Y 178.463,Z 373.256,A -85,B 0,C 180,E1 -22551.963,E2 -22551.963} C_VEL
LIN {X 0,Y 178.49,Z 373.25,A -85,B 0,C 180,E1 -22556.548,E2 -22556.548} C_VEL
LIN {X 0,Y 178.523,Z 373.248,A -85,B 0,C 180,E1 -22560.007,E2 -22560.007} C_VEL
LIN {X 0,Y 178.535,Z 373.243,A -85,B 0,C 180,E1 -22564.876,E2 -22564.876} C_VEL
LIN {X 0,Y 178.624,Z 373.229,A -85,B 0,C 180,E1 -22570.784,E2 -22570.784} C_VEL
LIN {X 0,Y 178.667,Z 373.23,A -85,B 0,C 180,E1 -22574.018,E2 -22574.018} C_VEL
LIN {X 0,Y 178.896,Z 373.197,A -85,B 0,C 180,E1 -22579.154,E2 -22579.154} C_VEL
LIN {X 0,Y 178.936,Z 373.196,A -85,B 0,C 180,E1 -22583.233,E2 -22583.233} C_VEL
LIN {X 0,Y 179.159,Z 373.167,A -85,B 0,C 180,E1 -22587.752,E2 -22587.752} C_VEL
LIN {X 0,Y 179.375,Z 373.141,A -85,B 0,C 180,E1 -22590,E2 -22590} C_VEL
LIN {X 0,Y 178.874,Z 373.195,A -85,B 0,C 180,E1 -22594.507,E2 -22594.507} C_VEL
LIN {X 0,Y 178.959,Z 373.193,A -85,B 0,C 180,E1 -22599.038,E2 -22599.038} C_VEL
LIN {X 0,Y 178.663,Z 373.23,A -85,B 0,C 180,E1 -22603.651,E2 -22603.651} C_VEL
LIN {X 0,Y 178.639,Z 373.235,A -85,B 0,C 180,E1 -22609.23,E2 -22609.23} C_VEL
LIN {X 0,Y 178.535,Z 373.247,A -85,B 0,C 180,E1 -22615.124,E2 -22615.124} C_VEL
LIN {X 0,Y 178.501,Z 373.251,A -85,B 0,C 180,E1 -22620.786,E2 -22620.786} C_VEL
LIN {X 0,Y 178.545,Z 373.392,A -85,B 0,C 180,E1 -22622.767,E2 -22622.767} C_VEL
LIN {X 0,Y 178.847,Z 374.564,A -85,B 0,C 180,E1 -22623.208,E2 -22623.208} C_VEL
LIN {X 0,Y 182.77,Z 387.868,A -85,B 0,C 180,E1 -22625.596,E2 -22625.596} C_VEL
LIN {X 0,Y 185.729,Z 399.054,A -85,B 0,C 180,E1 -22627.944,E2 -22627.944} C_VEL
LIN {X 0,Y 186.438,Z 403.327,A -85,B 0,C 180,E1 -22628.912,E2 -22628.912} C_VEL
LIN {X 0,Y 184.449,Z 414.86,A -85,B 0,C 180,E1 -22631.603,E2 -22631.603} C_VEL
LIN {X 0,Y 182.683,Z 425.193,A -85,B 0,C 180,E1 -22634.625,E2 -22634.625} C_VEL
LIN {X 0,Y 181.096,Z 434.58,A -85,B 0,C 180,E1 -22638.043,E2 -22638.043} C_VEL
LIN {X 0,Y 180.002,Z 441.891,A -85,B 0,C 180,E1 -22641.339,E2 -22641.339} C_VEL
LIN {X 0,Y 179.173,Z 449.101,A -85,B 0,C 180,E1 -22645.457,E2 -22645.457} C_VEL
LIN {X 0,Y 178.928,Z 454.308,A -85,B 0,C 180,E1 -22649.295,E2 -22649.295} C_VEL
LIN {X 0,Y 179.242,Z 458.213,A -85,B 0,C 180,E1 -22653.184,E2 -22653.184} C_VEL
LIN {X 0,Y 180.218,Z 460.902,A -85,B 0,C 180,E1 -22657.047,E2 -22657.047} C_VEL
LIN {X 0,Y 181.207,Z 462.062,A -85,B 0,C 180,E1 -22659.57,E2 -22659.57} C_VEL
LIN {X 0,Y 183.28,Z 462.888,A -85,B 0,C 180,E1 -22663.46,E2 -22663.46} C_VEL
LIN {X 0,Y 186.74,Z 462.246,A -85,B 0,C 180,E1 -22668.095,E2 -22668.095} C_VEL
LIN {X 0,Y 191.32,Z 459.752,A -85,B 0,C 180,E1 -22672.658,E2 -22672.658} C_VEL
LIN {X 0,Y 195.396,Z 456.623,A -85,B 0,C 180,E1 -22675.875,E2 -22675.875} C_VEL
LIN {X 0,Y 200,Z 452.339,A -85,B 0,C 180,E1 -22678.993,E2 -22678.993} C_VEL
LIN {X 0,Y 205.135,Z 446.736,A -85,B 0,C 180,E1 -22681.963,E2 -22681.963} C_VEL
LIN {X 0,Y 210.676,Z 439.588,A -85,B 0,C 180,E1 -22684.784,E2 -22684.784} C_VEL
LIN {X 0,Y 211.648,Z 437.608,A -85,B 0,C 180,E1 -22685.717,E2 -22685.717} C_VEL
LIN {X 0,Y 212.392,Z 432.938,A -85,B 0,C 180,E1 -22688.564,E2 -22688.564} C_VEL
LIN {X 0,Y 212.403,Z 427.399,A -85,B 0,C 180,E1 -22692.42,E2 -22692.42} C_VEL
LIN {X 0,Y 211.99,Z 423.181,A -85,B 0,C 180,E1 -22695.971,E2 -22695.971} C_VEL
LIN {X 0,Y 211.578,Z 421.971,A -85,B 0,C 180,E1 -22697.395,E2 -22697.395} C_VEL
LIN {X 0,Y 210.021,Z 420.336,A -85,B 0,C 180,E1 -22701.598,E2 -22701.598} C_VEL
LIN {X 0,Y 209.19,Z 420.087,A -85,B 0,C 180,E1 -22704.896,E2 -22704.896} C_VEL
LIN {X 0,Y 208.459,Z 421.474,A -85,B 0,C 180,E1 -22708.772,E2 -22708.772} C_VEL
LIN {X 0,Y 208.393,Z 424.167,A -85,B 0,C 180,E1 -22712.656,E2 -22712.656} C_VEL
LIN {X 0,Y 209.035,Z 427.55,A -85,B 0,C 180,E1 -22716.207,E2 -22716.207} C_VEL
LIN {X 0,Y 209.302,Z 429.511,A -85,B 0,C 180,E1 -22717.64,E2 -22717.64} C_VEL
LIN {X 0,Y 209.975,Z 436.021,A -85,B 0,C 180,E1 -22721.507,E2 -22721.507} C_VEL
LIN {X 0,Y 210.139,Z 438.266,A -85,B 0,C 180,E1 -22722.628,E2 -22722.628} C_VEL
LIN {X 0,Y 208.732,Z 445.427,A -85,B 0,C 180,E1 -22725.005,E2 -22725.005} C_VEL
LIN {X 0,Y 206.358,Z 454.344,A -85,B 0,C 180,E1 -22727.797,E2 -22727.797} C_VEL
LIN {X 0,Y 203.604,Z 462.708,A -85,B 0,C 180,E1 -22730.452,E2 -22730.452} C_VEL
LIN {X 0,Y 200.063,Z 471.315,A -85,B 0,C 180,E1 -22733.332,E2 -22733.332} C_VEL
LIN {X 0,Y 195.951,Z 479.225,A -85,B 0,C 180,E1 -22736.227,E2 -22736.227} C_VEL
LIN {X 0,Y 191.12,Z 487.078,A -85,B 0,C 180,E1 -22739.628,E2 -22739.628} C_VEL
LIN {X 0,Y 186.631,Z 493.518,A -85,B 0,C 180,E1 -22743.136,E2 -22743.136} C_VEL
LIN {X 0,Y 182.277,Z 499.278,A -85,B 0,C 180,E1 -22747.322,E2 -22747.322} C_VEL
LIN {X 0,Y 180.554,Z 501.608,A -85,B 0,C 180,E1 -22749.494,E2 -22749.494} C_VEL
LIN {X 0,Y 178.246,Z 505.136,A -85,B 0,C 180,E1 -22753.979,E2 -22753.979} C_VEL
LIN {X 0,Y 177.234,Z 507.258,A -85,B 0,C 180,E1 -22758.565,E2 -22758.565} C_VEL
LIN {X 0,Y 177.56,Z 508.01,A -85,B 0,C 180,E1 -22763.181,E2 -22763.181} C_VEL
LIN {X 0,Y 178.704,Z 507.229,A -85,B 0,C 180,E1 -22767.746,E2 -22767.746} C_VEL
LIN {X 0,Y 179.434,Z 506.226,A -85,B 0,C 180,E1 -22770,E2 -22770} C_VEL
LIN {X 0,Y 178.798,Z 503.443,A -85,B 0,C 180,E1 -22773.38,E2 -22773.38} C_VEL
LIN {X 0,Y 178.256,Z 499.465,A -85,B 0,C 180,E1 -22776.793,E2 -22776.793} C_VEL
LIN {X 0,Y 178.082,Z 496.833,A -85,B 0,C 180,E1 -22778.624,E2 -22778.624} C_VEL
LIN {X 0,Y 177.377,Z 494.038,A -85,B 0,C 180,E1 -22780.29,E2 -22780.29} C_VEL
LIN {X 0,Y 174.7,Z 488.748,A -85,B 0,C 180,E1 -22782.888,E2 -22782.888} C_VEL
LIN {X 0,Y 172.416,Z 482.813,A -85,B 0,C 180,E1 -22785.419,E2 -22785.419} C_VEL
LIN {X 0,Y 172.353,Z 479.005,A -85,B 0,C 180,E1 -22786.93,E2 -22786.93} C_VEL
LIN {X 0,Y 173.481,Z 471.743,A -85,B 0,C 180,E1 -22789.525,E2 -22789.525} C_VEL
LIN {X 0,Y 173.496,Z 463.407,A -85,B 0,C 180,E1 -22792.005,E2 -22792.005} C_VEL
LIN {X 0,Y 173.496,Z 451.835,A -85,B 0,C 180,E1 -22794.851,E2 -22794.851} C_VEL
LIN {X 0,Y 173.45,Z 441.472,A -85,B 0,C 180,E1 -22796.948,E2 -22796.948} C_VEL
LIN {X 0,Y 173.222,Z 429.14,A -85,B 0,C 180,E1 -22798.982,E2 -22798.982} C_VEL
LIN {X 0,Y 172.804,Z 415.184,A -85,B 0,C 180,E1 -22800.746,E2 -22800.746} C_VEL
LIN {X 0,Y 172.4,Z 402.647,A -85,B 0,C 180,E1 -22802.001,E2 -22802.001} C_VEL
LIN {X 0,Y 172.79,Z 400.619,A -85,B 0,C 180,E1 -22803.304,E2 -22803.304} C_VEL
LIN {X 0,Y 174.761,Z 393.6,A -85,B 0,C 180,E1 -22808.559,E2 -22808.559} C_VEL
LIN {X 0,Y 174.978,Z 391.345,A -85,B 0,C 180,E1 -22810.258,E2 -22810.258} C_VEL
LIN {X 0,Y 174.149,Z 387.334,A -85,B 0,C 180,E1 -22813.413,E2 -22813.413} C_VEL
LIN {X 0,Y 172.881,Z 381.523,A -85,B 0,C 180,E1 -22818.138,E2 -22818.138} C_VEL
LIN {X 0,Y 171.708,Z 375.148,A -85,B 0,C 180,E1 -22823.595,E2 -22823.595} C_VEL
LIN {X 0,Y 171.505,Z 374.169,A -85,B 0,C 180,E1 -22824.632,E2 -22824.632} C_VEL
LIN {X 0,Y 171.446,Z 374.126,A -85,B 0,C 180,E1 -22830.534,E2 -22830.534} C_VEL
LIN {X 0,Y 171.44,Z 374.127,A -85,B 0,C 180,E1 -22835.799,E2 -22835.799} C_VEL
LIN {X 0,Y 171.542,Z 374.117,A -85,B 0,C 180,E1 -22840.867,E2 -22840.867} C_VEL
LIN {X 0,Y 171.554,Z 374.107,A -85,B 0,C 180,E1 -22845.771,E2 -22845.771} C_VEL
LIN {X 0,Y 171.839,Z 374.077,A -85,B 0,C 180,E1 -22850.584,E2 -22850.584} C_VEL
LIN {X 0,Y 171.803,Z 374.081,A -85,B 0,C 180,E1 -22855.307,E2 -22855.307} C_VEL
LIN {X 0,Y 172.327,Z 374.018,A -85,B 0,C 180,E1 -22860,E2 -22860} C_VEL
LIN {X 0,Y 171.813,Z 374.08,A -85,B 0,C 180,E1 -22864.693,E2 -22864.693} C_VEL
LIN {X 0,Y 171.869,Z 374.075,A -85,B 0,C 180,E1 -22869.414,E2 -22869.414} C_VEL
LIN {X 0,Y 171.589,Z 374.106,A -85,B 0,C 180,E1 -22874.226,E2 -22874.226} C_VEL
LIN {X 0,Y 171.541,Z 374.115,A -85,B 0,C 180,E1 -22879.562,E2 -22879.562} C_VEL
LIN {X 0,Y 171.466,Z 374.125,A -85,B 0,C 180,E1 -22885.617,E2 -22885.617} C_VEL
LIN {X 0,Y 171.439,Z 374.127,A -85,B 0,C 180,E1 -22890.587,E2 -22890.587} C_VEL
LIN {X 0,Y 171.405,Z 374.133,A -85,B 0,C 180,E1 -22895.032,E2 -22895.032} C_VEL
LIN {X 0,Y 171.393,Z 374.132,A -85,B 0,C 180,E1 -22898.824,E2 -22898.824} C_VEL
LIN {X 0,Y 171.342,Z 374.141,A -85,B 0,C 180,E1 -22904.21,E2 -22904.21} C_VEL
LIN {X 0,Y 171.346,Z 374.139,A -85,B 0,C 180,E1 -22908.986,E2 -22908.986} C_VEL
LIN {X 0,Y 171.412,Z 374.133,A -85,B 0,C 180,E1 -22912.049,E2 -22912.049} C_VEL
LIN {X 0,Y 171.41,Z 374.128,A -85,B 0,C 180,E1 -22915.087,E2 -22915.087} C_VEL
LIN {X 0,Y 171.449,Z 374.126,A -85,B 0,C 180,E1 -22920.535,E2 -22920.535} C_VEL
LIN {X 0,Y 171.458,Z 374.127,A -85,B 0,C 180,E1 -22925.802,E2 -22925.802} C_VEL
LIN {X 0,Y 171.58,Z 374.107,A -85,B 0,C 180,E1 -22930.872,E2 -22930.872} C_VEL
LIN {X 0,Y 171.611,Z 374.109,A -85,B 0,C 180,E1 -22935.776,E2 -22935.776} C_VEL
LIN {X 0,Y 171.912,Z 374.067,A -85,B 0,C 180,E1 -22940.589,E2 -22940.589} C_VEL
LIN {X 0,Y 171.83,Z 374.082,A -85,B 0,C 180,E1 -22945.308,E2 -22945.308} C_VEL
LIN {X 0,Y 172.337,Z 374.018,A -85,B 0,C 180,E1 -22950,E2 -22950} C_VEL
LIN {X 0,Y 171.823,Z 374.073,A -85,B 0,C 180,E1 -22954.692,E2 -22954.692} C_VEL
LIN {X 0,Y 171.888,Z 374.075,A -85,B 0,C 180,E1 -22959.413,E2 -22959.413} C_VEL
LIN {X 0,Y 171.583,Z 374.111,A -85,B 0,C 180,E1 -22964.226,E2 -22964.226} C_VEL
LIN {X 0,Y 171.559,Z 374.115,A -85,B 0,C 180,E1 -22969.574,E2 -22969.574} C_VEL
LIN {X 0,Y 171.469,Z 374.125,A -85,B 0,C 180,E1 -22975.615,E2 -22975.615} C_VEL
LIN {X 0,Y 171.467,Z 374.126,A -85,B 0,C 180,E1 -22981.284,E2 -22981.284} C_VEL
LIN {X 0,Y 171.519,Z 374.347,A -85,B 0,C 180,E1 -22982.186,E2 -22982.186} C_VEL
LIN {X 0,Y 171.872,Z 375.772,A -85,B 0,C 180,E1 -22982.632,E2 -22982.632} C_VEL
LIN {X 0,Y 175.658,Z 388.474,A -85,B 0,C 180,E1 -22985.009,E2 -22985.009} C_VEL
LIN {X 0,Y 178.576,Z 399.72,A -85,B 0,C 180,E1 -22987.453,E2 -22987.453} C_VEL
LIN {X 0,Y 179.491,Z 403.909,A -85,B 0,C 180,E1 -22988.454,E2 -22988.454} C_VEL
LIN {X 0,Y 177.485,Z 415.357,A -85,B 0,C 180,E1 -22991.205,E2 -22991.205} C_VEL
LIN {X 0,Y 175.825,Z 424.756,A -85,B 0,C 180,E1 -22993.988,E2 -22993.988} C_VEL
LIN {X 0,Y 174.17,Z 434.265,A -85,B 0,C 180,E1 -22997.477,E2 -22997.477} C_VEL
LIN {X 0,Y 173.118,Z 440.952,A -85,B 0,C 180,E1 -23000.472,E2 -23000.472} C_VEL
LIN {X 0,Y 172.361,Z 446.788,A -85,B 0,C 180,E1 -23003.634,E2 -23003.634} C_VEL
LIN {X 0,Y 171.872,Z 453.084,A -85,B 0,C 180,E1 -23007.888,E2 -23007.888} C_VEL
LIN {X 0,Y 172.029,Z 457.664,A -85,B 0,C 180,E1 -23011.978,E2 -23011.978} C_VEL
LIN {X 0,Y 172.821,Z 460.922,A -85,B 0,C 180,E1 -23016.005,E2 -23016.005} C_VEL
LIN {X 0,Y 173.703,Z 462.45,A -85,B 0,C 180,E1 -23018.645,E2 -23018.645} C_VEL
LIN {X 0,Y 174.918,Z 463.459,A -85,B 0,C 180,E1 -23021.251,E2 -23021.251} C_VEL
LIN {X 0,Y 176.365,Z 463.975,A -85,B 0,C 180,E1 -23023.803,E2 -23023.803} C_VEL
LIN {X 0,Y 179.552,Z 463.794,A -85,B 0,C 180,E1 -23028.104,E2 -23028.104} C_VEL
LIN {X 0,Y 182.374,Z 462.739,A -85,B 0,C 180,E1 -23031.133,E2 -23031.133} C_VEL
LIN {X 0,Y 184.936,Z 461.397,A -85,B 0,C 180,E1 -23033.454,E2 -23033.454} C_VEL
LIN {X 0,Y 189.967,Z 457.92,A -85,B 0,C 180,E1 -23037.267,E2 -23037.267} C_VEL
LIN {X 0,Y 194.131,Z 454.338,A -85,B 0,C 180,E1 -23040,E2 -23040} C_VEL
LIN {X 0,Y 199.542,Z 448.93,A -85,B 0,C 180,E1 -23043.028,E2 -23043.028} C_VEL
LIN {X 0,Y 205.382,Z 442.156,A -85,B 0,C 180,E1 -23045.892,E2 -23045.892} C_VEL
LIN {X 0,Y 206.203,Z 440.393,A -85,B 0,C 180,E1 -23046.851,E2 -23046.851} C_VEL
LIN {X 0,Y 206.874,Z 437.468,A -85,B 0,C 180,E1 -23048.794,E2 -23048.794} C_VEL
LIN {X 0,Y 207.371,Z 432.302,A -85,B 0,C 180,E1 -23052.726,E2 -23052.726} C_VEL
LIN {X 0,Y 207.426,Z 428.981,A -85,B 0,C 180,E1 -23055.727,E2 -23055.727} C_VEL
LIN {X 0,Y 206.946,Z 427.295,A -85,B 0,C 180,E1 -23058.034,E2 -23058.034} C_VEL
LIN {X 0,Y 205.779,Z 426.077,A -85,B 0,C 180,E1 -23062.067,E2 -23062.067} C_VEL
LIN {X 0,Y 205.35,Z 425.93,A -85,B 0,C 180,E1 -23064.249,E2 -23064.249} C_VEL
LIN {X 0,Y 204.8,Z 426.621,A -85,B 0,C 180,E1 -23066.848,E2 -23066.848} C_VEL
LIN {X 0,Y 204.391,Z 428.69,A -85,B 0,C 180,E1 -23070.728,E2 -23070.728} C_VEL
LIN {X 0,Y 204.805,Z 432.959,A -85,B 0,C 180,E1 -23075.688,E2 -23075.688} C_VEL
LIN {X 0,Y 204.958,Z 436.328,A -85,B 0,C 180,E1 -23078.114,E2 -23078.114} C_VEL
LIN {X 0,Y 205.243,Z 441.274,A -85,B 0,C 180,E1 -23081.122,E2 -23081.122} C_VEL
LIN {X 0,Y 205.192,Z 443.128,A -85,B 0,C 180,E1 -23082.06,E2 -23082.06} C_VEL
LIN {X 0,Y 202.474,Z 452.466,A -85,B 0,C 180,E1 -23085.246,E2 -23085.246} C_VEL
LIN {X 0,Y 198.903,Z 462.305,A -85,B 0,C 180,E1 -23088.578,E2 -23088.578} C_VEL
LIN {X 0,Y 195.088,Z 470.827,A -85,B 0,C 180,E1 -23091.581,E2 -23091.581} C_VEL
LIN {X 0,Y 190.851,Z 478.498,A -85,B 0,C 180,E1 -23094.551,E2 -23094.551} C_VEL
LIN {X 0,Y 185.678,Z 486.196,A -85,B 0,C 180,E1 -23098.002,E2 -23098.002} C_VEL
LIN {X 0,Y 181.638,Z 491.693,A -85,B 0,C 180,E1 -23101.077,E2 -23101.077} C_VEL
LIN {X 0,Y 176.755,Z 497.574,A -85,B 0,C 180,E1 -23105.324,E2 -23105.324} C_VEL
LIN {X 0,Y 173.851,Z 500.982,A -85,B 0,C 180,E1 -23108.665,E2 -23108.665} C_VEL
LIN {X 0,Y 171.385,Z 504.289,A -85,B 0,C 180,E1 -23113.319,E2 -23113.319} C_VEL
LIN {X 0,Y 170.245,Z 506.234,A -85,B 0,C 180,E1 -23118.088,E2 -23118.088} C_VEL
LIN {X 0,Y 170.504,Z 506.767,A -85,B 0,C 180,E1 -23122.897,E2 -23122.897} C_VEL
LIN {X 0,Y 171.704,Z 505.819,A -85,B 0,C 180,E1 -23127.654,E2 -23127.654} C_VEL
LIN {X 0,Y 172.452,Z 504.744,A -85,B 0,C 180,E1 -23130,E2 -23130} C_VEL
LIN {X 0,Y 171.78,Z 501.803,A -85,B 0,C 180,E1 -23133.518,E2 -23133.518} C_VEL
LIN {X 0,Y 171.227,Z 497.662,A -85,B 0,C 180,E1 -23137.073,E2 -23137.073} C_VEL
LIN {X 0,Y 171.15,Z 491.299,A -85,B 0,C 180,E1 -23141.187,E2 -23141.187} C_VEL
LIN {X 0,Y 171.695,Z 484.05,A -85,B 0,C 180,E1 -23144.823,E2 -23144.823} C_VEL
LIN {X 0,Y 172.353,Z 479.005,A -85,B 0,C 180,E1 -23146.93,E2 -23146.93} C_VEL
LIN {X 0,Y 172.437,Z 476.421,A -85,B 0,C 180,E1 -23147.901,E2 -23147.901} C_VEL
LIN {X 0,Y 171.908,Z 473.695,A -85,B 0,C 180,E1 -23148.838,E2 -23148.838} C_VEL
LIN {X 0,Y 169.801,Z 468.155,A -85,B 0,C 180,E1 -23150.619,E2 -23150.619} C_VEL
LIN {X 0,Y 167.021,Z 460.744,A -85,B 0,C 180,E1 -23152.77,E2 -23152.77} C_VEL
LIN {X 0,Y 166.418,Z 455.977,A -85,B 0,C 180,E1 -23154.028,E2 -23154.028} C_VEL
LIN {X 0,Y 166.422,Z 444.513,A -85,B 0,C 180,E1 -23156.659,E2 -23156.659} C_VEL
LIN {X 0,Y 166.309,Z 432.317,A -85,B 0,C 180,E1 -23158.902,E2 -23158.902} C_VEL
LIN {X 0,Y 166.038,Z 419.849,A -85,B 0,C 180,E1 -23160.726,E2 -23160.726} C_VEL
LIN {X 0,Y 165.591,Z 405.978,A -85,B 0,C 180,E1 -23162.256,E2 -23162.256} C_VEL
LIN {X 0,Y 165.506,Z 401.577,A -85,B 0,C 180,E1 -23162.765,E2 -23162.765} C_VEL
LIN {X 0,Y 167.344,Z 394.929,A -85,B 0,C 180,E1 -23167.811,E2 -23167.811} C_VEL
LIN {X 0,Y 167.917,Z 392.231,A -85,B 0,C 180,E1 -23169.932,E2 -23169.932} C_VEL
LIN {X 0,Y 167.124,Z 388.179,A -85,B 0,C 180,E1 -23173.227,E2 -23173.227} C_VEL
LIN {X 0,Y 165.707,Z 381.708,A -85,B 0,C 180,E1 -23178.752,E2 -23178.752} C_VEL
LIN {X 0,Y 164.5,Z 375.3,A -85,B 0,C 180,E1 -23184.494,E2 -23184.494} C_VEL
LIN {X 0,Y 164.37,Z 375.011,A -85,B 0,C 180,E1 -23186.231,E2 -23186.231} C_VEL
LIN {X 0,Y 164.39,Z 375.008,A -85,B 0,C 180,E1 -23189.134,E2 -23189.134} C_VEL
LIN {X 0,Y 164.403,Z 375.006,A -85,B 0,C 180,E1 -23194.692,E2 -23194.692} C_VEL
LIN {X 0,Y 164.436,Z 375,A -85,B 0,C 180,E1 -23200.095,E2 -23200.095} C_VEL
LIN {X 0,Y 164.482,Z 374.99,A -85,B 0,C 180,E1 -23205.145,E2 -23205.145} C_VEL
LIN {X 0,Y 164.76,Z 374.958,A -85,B 0,C 180,E1 -23210.176,E2 -23210.176} C_VEL
LIN {X 0,Y 164.82,Z 374.954,A -85,B 0,C 180,E1 -23212.65,E2 -23212.65} C_VEL
LIN {X 0,Y 165.039,Z 374.923,A -85,B 0,C 180,E1 -23217.559,E2 -23217.559} C_VEL
LIN {X 0,Y 165.29,Z 374.894,A -85,B 0,C 180,E1 -23220,E2 -23220} C_VEL
LIN {X 0,Y 164.762,Z 374.957,A -85,B 0,C 180,E1 -23224.894,E2 -23224.894} C_VEL
LIN {X 0,Y 164.841,Z 374.95,A -85,B 0,C 180,E1 -23227.348,E2 -23227.348} C_VEL
LIN {X 0,Y 164.747,Z 374.961,A -85,B 0,C 180,E1 -23231.146,E2 -23231.146} C_VEL
LIN {X 0,Y 164.481,Z 374.995,A -85,B 0,C 180,E1 -23237.403,E2 -23237.403} C_VEL
LIN {X 0,Y 164.471,Z 374.996,A -85,B 0,C 180,E1 -23239.989,E2 -23239.989} C_VEL
LIN {X 0,Y 164.391,Z 375.008,A -85,B 0,C 180,E1 -23246.134,E2 -23246.134} C_VEL
LIN {X 0,Y 164.373,Z 375.006,A -85,B 0,C 180,E1 -23251.229,E2 -23251.229} C_VEL
LIN {X 0,Y 164.314,Z 375.014,A -85,B 0,C 180,E1 -23256.784,E2 -23256.784} C_VEL
LIN {X 0,Y 164.307,Z 375.015,A -85,B 0,C 180,E1 -23259.911,E2 -23259.911} C_VEL
LIN {X 0,Y 164.305,Z 375.017,A -85,B 0,C 180,E1 -23263.353,E2 -23263.353} C_VEL
LIN {X 0,Y 164.291,Z 375.016,A -85,B 0,C 180,E1 -23266.809,E2 -23266.809} C_VEL
LIN {X 0,Y 164.305,Z 375.019,A -85,B 0,C 180,E1 -23270.348,E2 -23270.348} C_VEL
LIN {X 0,Y 164.342,Z 375.009,A -85,B 0,C 180,E1 -23274.343,E2 -23274.343} C_VEL
LIN {X 0,Y 164.391,Z 375.007,A -85,B 0,C 180,E1 -23279.136,E2 -23279.136} C_VEL
LIN {X 0,Y 164.417,Z 375.002,A -85,B 0,C 180,E1 -23284.695,E2 -23284.695} C_VEL
LIN {X 0,Y 164.485,Z 374.992,A -85,B 0,C 180,E1 -23290.052,E2 -23290.052} C_VEL
LIN {X 0,Y 164.555,Z 374.987,A -85,B 0,C 180,E1 -23295.152,E2 -23295.152} C_VEL
LIN {X 0,Y 164.854,Z 374.946,A -85,B 0,C 180,E1 -23300.182,E2 -23300.182} C_VEL
LIN {X 0,Y 164.78,Z 374.959,A -85,B 0,C 180,E1 -23305.107,E2 -23305.107} C_VEL
LIN {X 0,Y 165.299,Z 374.895,A -85,B 0,C 180,E1 -23310,E2 -23310} C_VEL
LIN {X 0,Y 164.773,Z 374.951,A -85,B 0,C 180,E1 -23314.893,E2 -23314.893} C_VEL
LIN {X 0,Y 164.851,Z 374.948,A -85,B 0,C 180,E1 -23317.348,E2 -23317.348} C_VEL
LIN {X 0,Y 164.743,Z 374.961,A -85,B 0,C 180,E1 -23321.131,E2 -23321.131} C_VEL
LIN {X 0,Y 164.499,Z 374.992,A -85,B 0,C 180,E1 -23327.401,E2 -23327.401} C_VEL
LIN {X 0,Y 164.476,Z 374.996,A -85,B 0,C 180,E1 -23329.988,E2 -23329.988} C_VEL
LIN {X 0,Y 164.393,Z 375.006,A -85,B 0,C 180,E1 -23336.133,E2 -23336.133} C_VEL
LIN {X 0,Y 164.448,Z 375.146,A -85,B 0,C 180,E1 -23341.436,E2 -23341.436} C_VEL
LIN {X 0,Y 164.744,Z 376.393,A -85,B 0,C 180,E1 -23341.926,E2 -23341.926} C_VEL
LIN {X 0,Y 168.407,Z 388.587,A -85,B 0,C 180,E1 -23344.289,E2 -23344.289} C_VEL
LIN {X 0,Y 171.122,Z 398.786,A -85,B 0,C 180,E1 -23346.548,E2 -23346.548} C_VEL
LIN {X 0,Y 172.499,Z 404.837,A -85,B 0,C 180,E1 -23348.04,E2 -23348.04} C_VEL
LIN {X 0,Y 170.383,Z 416.525,A -85,B 0,C 180,E1 -23350.959,E2 -23350.959} C_VEL
LIN {X 0,Y 168.606,Z 426.355,A -85,B 0,C 180,E1 -23354.025,E2 -23354.025} C_VEL
LIN {X 0,Y 166.947,Z 435.701,A -85,B 0,C 180,E1 -23357.658,E2 -23357.658} C_VEL
LIN {X 0,Y 165.818,Z 443.311,A -85,B 0,C 180,E1 -23361.306,E2 -23361.306} C_VEL
LIN {X 0,Y 165.036,Z 449.769,A -85,B 0,C 180,E1 -23365.138,E2 -23365.138} C_VEL
LIN {X 0,Y 164.769,Z 455.186,A -85,B 0,C 180,E1 -23369.213,E2 -23369.213} C_VEL
LIN {X 0,Y 165.127,Z 459.409,A -85,B 0,C 180,E1 -23373.35,E2 -23373.35} C_VEL
LIN {X 0,Y 166.46,Z 462.918,A -85,B 0,C 180,E1 -23378.252,E2 -23378.252} C_VEL
LIN {X 0,Y 168.858,Z 464.844,A -85,B 0,C 180,E1 -23383.187,E2 -23383.187} C_VEL
LIN {X 0,Y 170.452,Z 465.244,A -85,B 0,C 180,E1 -23385.677,E2 -23385.677} C_VEL
LIN {X 0,Y 172.443,Z 465.156,A -85,B 0,C 180,E1 -23388.242,E2 -23388.242} C_VEL
LIN {X 0,Y 174.721,Z 464.634,A -85,B 0,C 180,E1 -23390.741,E2 -23390.741} C_VEL
LIN {X 0,Y 177.259,Z 463.672,A -85,B 0,C 180,E1 -23393.169,E2 -23393.169} C_VEL
LIN {X 0,Y 180.096,Z 462.188,A -85,B 0,C 180,E1 -23395.524,E2 -23395.524} C_VEL
LIN {X 0,Y 184.928,Z 459.031,A -85,B 0,C 180,E1 -23398.911,E2 -23398.911} C_VEL
LIN {X 0,Y 190.226,Z 454.766,A -85,B 0,C 180,E1 -23402.117,E2 -23402.117} C_VEL
LIN {X 0,Y 196.041,Z 449.198,A -85,B 0,C 180,E1 -23405.143,E2 -23405.143} C_VEL
LIN {X 0,Y 200.056,Z 444.709,A -85,B 0,C 180,E1 -23407.063,E2 -23407.063} C_VEL
LIN {X 0,Y 201.227,Z 441.867,A -85,B 0,C 180,E1 -23409.043,E2 -23409.043} C_VEL
LIN {X 0,Y 201.989,Z 438.21,A -85,B 0,C 180,E1 -23412.05,E2 -23412.05} C_VEL
LIN {X 0,Y 202.455,Z 434.94,A -85,B 0,C 180,E1 -23415.091,E2 -23415.091} C_VEL
LIN {X 0,Y 202.547,Z 433.97,A -85,B 0,C 180,E1 -23416.116,E2 -23416.116} C_VEL
LIN {X 0,Y 202.301,Z 432.639,A -85,B 0,C 180,E1 -23418.22,E2 -23418.22} C_VEL
LIN {X 0,Y 201.746,Z 431.985,A -85,B 0,C 180,E1 -23420.387,E2 -23420.387} C_VEL
LIN {X 0,Y 201.321,Z 431.63,A -85,B 0,C 180,E1 -23422.582,E2 -23422.582} C_VEL
LIN {X 0,Y 200.879,Z 431.75,A -85,B 0,C 180,E1 -23424.824,E2 -23424.824} C_VEL
LIN {X 0,Y 200.285,Z 433.195,A -85,B 0,C 180,E1 -23428.69,E2 -23428.69} C_VEL
LIN {X 0,Y 200.073,Z 435.871,A -85,B 0,C 180,E1 -23432.538,E2 -23432.538} C_VEL
LIN {X 0,Y 200.339,Z 438.348,A -85,B 0,C 180,E1 -23435.321,E2 -23435.321} C_VEL
LIN {X 0,Y 200.286,Z 441.843,A -85,B 0,C 180,E1 -23437.934,E2 -23437.934} C_VEL
LIN {X 0,Y 200.257,Z 446.054,A -85,B 0,C 180,E1 -23440.615,E2 -23440.615} C_VEL
LIN {X 0,Y 199.945,Z 447.716,A -85,B 0,C 180,E1 -23441.398,E2 -23441.398} C_VEL
LIN {X 0,Y 196.885,Z 456.068,A -85,B 0,C 180,E1 -23444.447,E2 -23444.447} C_VEL
LIN {X 0,Y 192.898,Z 465.207,A -85,B 0,C 180,E1 -23447.762,E2 -23447.762} C_VEL
LIN {X 0,Y 188.083,Z 474.242,A -85,B 0,C 180,E1 -23451.254,E2 -23451.254} C_VEL
LIN {X 0,Y 183.525,Z 481.231,A -85,B 0,C 180,E1 -23454.269,E2 -23454.269} C_VEL
LIN {X 0,Y 178.234,Z 488.167,A -85,B 0,C 180,E1 -23457.838,E2 -23457.838} C_VEL
LIN {X 0,Y 172.713,Z 494.544,A -85,B 0,C 180,E1 -23462.099,E2 -23462.099} C_VEL
LIN {X 0,Y 169.198,Z 498.297,A -85,B 0,C 180,E1 -23465.458,E2 -23465.458} C_VEL
LIN {X 0,Y 167.199,Z 500.352,A -85,B 0,C 180,E1 -23467.772,E2 -23467.772} C_VEL
LIN {X 0,Y 164.553,Z 503.447,A -85,B 0,C 180,E1 -23472.605,E2 -23472.605} C_VEL
LIN {X 0,Y 163.283,Z 505.136,A -85,B 0,C 180,E1 -23477.573,E2 -23477.573} C_VEL
LIN {X 0,Y 163.473,Z 505.487,A -85,B 0,C 180,E1 -23482.59,E2 -23482.59} C_VEL
LIN {X 0,Y 164.694,Z 504.412,A -85,B 0,C 180,E1 -23487.554,E2 -23487.554} C_VEL
LIN {X 0,Y 165.462,Z 503.214,A -85,B 0,C 180,E1 -23490,E2 -23490} C_VEL
LIN {X 0,Y 164.76,Z 500.094,A -85,B 0,C 180,E1 -23493.668,E2 -23493.668} C_VEL
LIN {X 0,Y 164.204,Z 495.735,A -85,B 0,C 180,E1 -23497.377,E2 -23497.377} C_VEL
LIN {X 0,Y 164.198,Z 489.016,A -85,B 0,C 180,E1 -23501.73,E2 -23501.73} C_VEL
LIN {X 0,Y 164.827,Z 481.629,A -85,B 0,C 180,E1 -23505.455,E2 -23505.455} C_VEL
LIN {X 0,Y 166.263,Z 472.45,A -85,B 0,C 180,E1 -23509.122,E2 -23509.122} C_VEL
LIN {X 0,Y 166.472,Z 465.102,A -85,B 0,C 180,E1 -23511.509,E2 -23511.509} C_VEL
LIN {X 0,Y 166.418,Z 455.977,A -85,B 0,C 180,E1 -23514.028,E2 -23514.028} C_VEL
LIN {X 0,Y 165.824,Z 451.21,A -85,B 0,C 180,E1 -23515.209,E2 -23515.209} C_VEL
LIN {X 0,Y 162.991,Z 443.323,A -85,B 0,C 180,E1 -23517.054,E2 -23517.054} C_VEL
LIN {X 0,Y 160.028,Z 435.172,A -85,B 0,C 180,E1 -23518.785,E2 -23518.785} C_VEL
LIN {X 0,Y 159.241,Z 429.902,A -85,B 0,C 180,E1 -23519.752,E2 -23519.752} C_VEL
LIN {X 0,Y 159.015,Z 417.117,A -85,B 0,C 180,E1 -23521.657,E2 -23521.657} C_VEL
LIN {X 0,Y 158.602,Z 400.956,A -85,B 0,C 180,E1 -23523.466,E2 -23523.466} C_VEL
LIN {X 0,Y 158.795,Z 399.824,A -85,B 0,C 180,E1 -23524.044,E2 -23524.044} C_VEL
LIN {X 0,Y 160.226,Z 395.137,A -85,B 0,C 180,E1 -23527.884,E2 -23527.884} C_VEL
LIN {X 0,Y 160.681,Z 393.34,A -85,B 0,C 180,E1 -23529.36,E2 -23529.36} C_VEL
LIN {X 0,Y 160.433,Z 390.364,A -85,B 0,C 180,E1 -23531.866,E2 -23531.866} C_VEL
LIN {X 0,Y 159.091,Z 384.72,A -85,B 0,C 180,E1 -23536.785,E2 -23536.785} C_VEL
LIN {X 0,Y 158.082,Z 379.552,A -85,B 0,C 180,E1 -23541.507,E2 -23541.507} C_VEL
LIN {X 0,Y 157.416,Z 375.925,A -85,B 0,C 180,E1 -23545.108,E2 -23545.108} C_VEL
LIN {X 0,Y 157.27,Z 375.892,A -85,B 0,C 180,E1 -23550.556,E2 -23550.556} C_VEL
LIN {X 0,Y 157.313,Z 375.89,A -85,B 0,C 180,E1 -23553.464,E2 -23553.464} C_VEL
LIN {X 0,Y 157.374,Z 375.88,A -85,B 0,C 180,E1 -23559.684,E2 -23559.684} C_VEL
LIN {X 0,Y 157.417,Z 375.874,A -85,B 0,C 180,E1 -23564.462,E2 -23564.462} C_VEL
LIN {X 0,Y 157.683,Z 375.84,A -85,B 0,C 180,E1 -23569.73,E2 -23569.73} C_VEL
LIN {X 0,Y 157.758,Z 375.833,A -85,B 0,C 180,E1 -23572.319,E2 -23572.319} C_VEL
LIN {X 0,Y 158.252,Z 375.771,A -85,B 0,C 180,E1 -23580,E2 -23580} C_VEL
LIN {X 0,Y 157.798,Z 375.827,A -85,B 0,C 180,E1 -23587.678,E2 -23587.678} C_VEL
LIN {X 0,Y 157.677,Z 375.841,A -85,B 0,C 180,E1 -23591.315,E2 -23591.315} C_VEL
LIN {X 0,Y 157.458,Z 375.869,A -85,B 0,C 180,E1 -23595.534,E2 -23595.534} C_VEL
LIN {X 0,Y 157.367,Z 375.877,A -85,B 0,C 180,E1 -23600.933,E2 -23600.933} C_VEL
LIN {X 0,Y 157.312,Z 375.889,A -85,B 0,C 180,E1 -23606.685,E2 -23606.685} C_VEL
LIN {X 0,Y 157.276,Z 375.894,A -85,B 0,C 180,E1 -23612.427,E2 -23612.427} C_VEL
LIN {X 0,Y 157.283,Z 375.891,A -85,B 0,C 180,E1 -23616.458,E2 -23616.458} C_VEL
LIN {X 0,Y 157.214,Z 375.903,A -85,B 0,C 180,E1 -23622.11,E2 -23622.11} C_VEL
LIN {X 0,Y 157.212,Z 375.899,A -85,B 0,C 180,E1 -23627.891,E2 -23627.891} C_VEL
LIN {X 0,Y 157.282,Z 375.891,A -85,B 0,C 180,E1 -23633.544,E2 -23633.544} C_VEL
LIN {X 0,Y 157.295,Z 375.893,A -85,B 0,C 180,E1 -23638.096,E2 -23638.096} C_VEL
LIN {X 0,Y 157.322,Z 375.882,A -85,B 0,C 180,E1 -23643.467,E2 -23643.467} C_VEL
LIN {X 0,Y 157.395,Z 375.877,A -85,B 0,C 180,E1 -23649.668,E2 -23649.668} C_VEL
LIN {X 0,Y 157.48,Z 375.868,A -85,B 0,C 180,E1 -23654.469,E2 -23654.469} C_VEL
LIN {X 0,Y 157.774,Z 375.827,A -85,B 0,C 180,E1 -23659.737,E2 -23659.737} C_VEL
LIN {X 0,Y 157.826,Z 375.825,A -85,B 0,C 180,E1 -23662.323,E2 -23662.323} C_VEL
LIN {X 0,Y 158.261,Z 375.771,A -85,B 0,C 180,E1 -23670,E2 -23670} C_VEL
LIN {X 0,Y 157.808,Z 375.827,A -85,B 0,C 180,E1 -23677.678,E2 -23677.678} C_VEL
LIN {X 0,Y 157.674,Z 375.841,A -85,B 0,C 180,E1 -23681.302,E2 -23681.302} C_VEL
LIN {X 0,Y 157.463,Z 375.87,A -85,B 0,C 180,E1 -23685.533,E2 -23685.533} C_VEL
LIN {X 0,Y 157.372,Z 375.88,A -85,B 0,C 180,E1 -23690.932,E2 -23690.932} C_VEL
LIN {X 0,Y 157.314,Z 375.889,A -85,B 0,C 180,E1 -23696.684,E2 -23696.684} C_VEL
LIN {X 0,Y 157.393,Z 376.001,A -85,B 0,C 180,E1 -23700.711,E2 -23700.711} C_VEL
LIN {X 0,Y 157.639,Z 377.001,A -85,B 0,C 180,E1 -23701.176,E2 -23701.176} C_VEL
LIN {X 0,Y 161.411,Z 389.471,A -85,B 0,C 180,E1 -23703.72,E2 -23703.72} C_VEL
LIN {X 0,Y 164.388,Z 400.935,A -85,B 0,C 180,E1 -23706.382,E2 -23706.382} C_VEL
LIN {X 0,Y 165.495,Z 405.719,A -85,B 0,C 180,E1 -23707.621,E2 -23707.621} C_VEL
LIN {X 0,Y 163.388,Z 417.053,A -85,B 0,C 180,E1 -23710.567,E2 -23710.567} C_VEL
LIN {X 0,Y 161.446,Z 427.535,A -85,B 0,C 180,E1 -23713.961,E2 -23713.961} C_VEL
LIN {X 0,Y 159.718,Z 437.098,A -85,B 0,C 180,E1 -23717.854,E2 -23717.854} C_VEL
LIN {X 0,Y 158.625,Z 444.66,A -85,B 0,C 180,E1 -23721.663,E2 -23721.663} C_VEL
LIN {X 0,Y 157.847,Z 451.76,A -85,B 0,C 180,E1 -23726.182,E2 -23726.182} C_VEL
LIN {X 0,Y 157.74,Z 457.215,A -85,B 0,C 180,E1 -23730.653,E2 -23730.653} C_VEL
LIN {X 0,Y 158.383,Z 461.305,A -85,B 0,C 180,E1 -23735.068,E2 -23735.068} C_VEL
LIN {X 0,Y 159.791,Z 464.136,A -85,B 0,C 180,E1 -23739.399,E2 -23739.399} C_VEL
LIN {X 0,Y 161.614,Z 465.687,A -85,B 0,C 180,E1 -23743.072,E2 -23743.072} C_VEL
LIN {X 0,Y 164.745,Z 466.447,A -85,B 0,C 180,E1 -23747.684,E2 -23747.684} C_VEL
LIN {X 0,Y 167.019,Z 466.276,A -85,B 0,C 180,E1 -23750.31,E2 -23750.31} C_VEL
LIN {X 0,Y 169.881,Z 465.549,A -85,B 0,C 180,E1 -23753.149,E2 -23753.149} C_VEL
LIN {X 0,Y 172.394,Z 464.549,A -85,B 0,C 180,E1 -23755.323,E2 -23755.323} C_VEL
LIN {X 0,Y 175.816,Z 462.865,A -85,B 0,C 180,E1 -23757.878,E2 -23757.878} C_VEL
LIN {X 0,Y 180.767,Z 459.737,A -85,B 0,C 180,E1 -23761.114,E2 -23761.114} C_VEL
LIN {X 0,Y 186.566,Z 455.229,A -85,B 0,C 180,E1 -23764.321,E2 -23764.321} C_VEL
LIN {X 0,Y 192.977,Z 449.282,A -85,B 0,C 180,E1 -23767.396,E2 -23767.396} C_VEL
LIN {X 0,Y 194.749,Z 447.383,A -85,B 0,C 180,E1 -23768.3,E2 -23768.3} C_VEL
LIN {X 0,Y 195.871,Z 444.888,A -85,B 0,C 180,E1 -23770.335,E2 -23770.335} C_VEL
LIN {X 0,Y 197.154,Z 440.612,A -85,B 0,C 180,E1 -23774.45,E2 -23774.45} C_VEL
LIN {X 0,Y 197.487,Z 438.798,A -85,B 0,C 180,E1 -23776.541,E2 -23776.541} C_VEL
LIN {X 0,Y 197.369,Z 437.701,A -85,B 0,C 180,E1 -23778.692,E2 -23778.692} C_VEL
LIN {X 0,Y 196.814,Z 437.116,A -85,B 0,C 180,E1 -23781.813,E2 -23781.813} C_VEL
LIN {X 0,Y 196.197,Z 437.435,A -85,B 0,C 180,E1 -23785.458,E2 -23785.458} C_VEL
LIN {X 0,Y 195.836,Z 438.302,A -85,B 0,C 180,E1 -23787.81,E2 -23787.81} C_VEL
LIN {X 0,Y 195.472,Z 441.475,A -85,B 0,C 180,E1 -23792.637,E2 -23792.637} C_VEL
LIN {X 0,Y 195.598,Z 443.659,A -85,B 0,C 180,E1 -23795.092,E2 -23795.092} C_VEL
LIN {X 0,Y 195.365,Z 447.031,A -85,B 0,C 180,E1 -23797.702,E2 -23797.702} C_VEL
LIN {X 0,Y 195.156,Z 449.746,A -85,B 0,C 180,E1 -23799.56,E2 -23799.56} C_VEL
LIN {X 0,Y 194.554,Z 451.95,A -85,B 0,C 180,E1 -23800.661,E2 -23800.661} C_VEL
LIN {X 0,Y 190.63,Z 460.617,A -85,B 0,C 180,E1 -23804.038,E2 -23804.038} C_VEL
LIN {X 0,Y 186.361,Z 468.767,A -85,B 0,C 180,E1 -23807.25,E2 -23807.25} C_VEL
LIN {X 0,Y 181.791,Z 476.109,A -85,B 0,C 180,E1 -23810.368,E2 -23810.368} C_VEL
LIN {X 0,Y 176.973,Z 482.632,A -85,B 0,C 180,E1 -23813.44,E2 -23813.44} C_VEL
LIN {X 0,Y 170.738,Z 489.829,A -85,B 0,C 180,E1 -23817.649,E2 -23817.649} C_VEL
LIN {X 0,Y 165.128,Z 495.521,A -85,B 0,C 180,E1 -23822.085,E2 -23822.085} C_VEL
LIN {X 0,Y 160.608,Z 499.705,A -85,B 0,C 180,E1 -23826.808,E2 -23826.808} C_VEL
LIN {X 0,Y 157.751,Z 502.526,A -85,B 0,C 180,E1 -23831.829,E2 -23831.829} C_VEL
LIN {X 0,Y 156.342,Z 504.029,A -85,B 0,C 180,E1 -23837.011,E2 -23837.011} C_VEL
LIN {X 0,Y 156.434,Z 504.202,A -85,B 0,C 180,E1 -23842.254,E2 -23842.254} C_VEL
LIN {X 0,Y 157.705,Z 502.899,A -85,B 0,C 180,E1 -23847.446,E2 -23847.446} C_VEL
LIN {X 0,Y 158.468,Z 501.628,A -85,B 0,C 180,E1 -23850,E2 -23850} C_VEL
LIN {X 0,Y 157.765,Z 498.341,A -85,B 0,C 180,E1 -23853.831,E2 -23853.831} C_VEL
LIN {X 0,Y 157.194,Z 493.775,A -85,B 0,C 180,E1 -23857.708,E2 -23857.708} C_VEL
LIN {X 0,Y 157.194,Z 487.907,A -85,B 0,C 180,E1 -23861.606,E2 -23861.606} C_VEL
LIN {X 0,Y 157.821,Z 480.511,A -85,B 0,C 180,E1 -23865.497,E2 -23865.497} C_VEL
LIN {X 0,Y 159.256,Z 471.315,A -85,B 0,C 180,E1 -23869.328,E2 -23869.328} C_VEL
LIN {X 0,Y 159.366,Z 464.693,A -85,B 0,C 180,E1 -23871.586,E2 -23871.586} C_VEL
LIN {X 0,Y 159.352,Z 453.612,A -85,B 0,C 180,E1 -23874.77,E2 -23874.77} C_VEL
LIN {X 0,Y 159.366,Z 442.592,A -85,B 0,C 180,E1 -23877.355,E2 -23877.355} C_VEL
LIN {X 0,Y 159.241,Z 429.902,A -85,B 0,C 180,E1 -23879.752,E2 -23879.752} C_VEL
LIN {X 0,Y 158.521,Z 424.604,A -85,B 0,C 180,E1 -23880.662,E2 -23880.662} C_VEL
LIN {X 0,Y 155.701,Z 415.97,A -85,B 0,C 180,E1 -23882.098,E2 -23882.098} C_VEL
LIN {X 0,Y 152.7,Z 407.173,A -85,B 0,C 180,E1 -23883.396,E2 -23883.396} C_VEL
LIN {X 0,Y 151.716,Z 401.613,A -85,B 0,C 180,E1 -23884.059,E2 -23884.059} C_VEL
LIN {X 0,Y 151.77,Z 399.663,A -85,B 0,C 180,E1 -23884.357,E2 -23884.357} C_VEL
LIN {X 0,Y 153.365,Z 394.266,A -85,B 0,C 180,E1 -23888.828,E2 -23888.828} C_VEL
LIN {X 0,Y 153.512,Z 391.55,A -85,B 0,C 180,E1 -23891.209,E2 -23891.209} C_VEL
LIN {X 0,Y 151.796,Z 384.349,A -85,B 0,C 180,E1 -23897.797,E2 -23897.797} C_VEL
LIN {X 0,Y 150.809,Z 379.242,A -85,B 0,C 180,E1 -23902.711,E2 -23902.711} C_VEL
LIN {X 0,Y 150.367,Z 376.814,A -85,B 0,C 180,E1 -23905.275,E2 -23905.275} C_VEL
LIN {X 0,Y 150.218,Z 376.771,A -85,B 0,C 180,E1 -23912.105,E2 -23912.105} C_VEL
LIN {X 0,Y 150.255,Z 376.762,A -85,B 0,C 180,E1 -23918.026,E2 -23918.026} C_VEL
LIN {X 0,Y 150.314,Z 376.761,A -85,B 0,C 180,E1 -23920.896,E2 -23920.896} C_VEL
LIN {X 0,Y 150.412,Z 376.739,A -85,B 0,C 180,E1 -23926.489,E2 -23926.489} C_VEL
LIN {X 0,Y 150.604,Z 376.72,A -85,B 0,C 180,E1 -23929.242,E2 -23929.242} C_VEL
LIN {X 0,Y 150.696,Z 376.712,A -85,B 0,C 180,E1 -23931.957,E2 -23931.957} C_VEL
LIN {X 0,Y 151.212,Z 376.648,A -85,B 0,C 180,E1 -23940,E2 -23940} C_VEL
LIN {X 0,Y 150.734,Z 376.707,A -85,B 0,C 180,E1 -23948.041,E2 -23948.041} C_VEL
LIN {X 0,Y 150.608,Z 376.722,A -85,B 0,C 180,E1 -23951.5,E2 -23951.5} C_VEL
LIN {X 0,Y 150.364,Z 376.754,A -85,B 0,C 180,E1 -23956.286,E2 -23956.286} C_VEL
LIN {X 0,Y 150.348,Z 376.752,A -85,B 0,C 180,E1 -23960.792,E2 -23960.792} C_VEL
LIN {X 0,Y 150.242,Z 376.768,A -85,B 0,C 180,E1 -23967.283,E2 -23967.283} C_VEL
LIN {X 0,Y 150.216,Z 376.774,A -85,B 0,C 180,E1 -23972.635,E2 -23972.635} C_VEL
LIN {X 0,Y 150.211,Z 376.77,A -85,B 0,C 180,E1 -23977.462,E2 -23977.462} C_VEL
LIN {X 0,Y 150.156,Z 376.78,A -85,B 0,C 180,E1 -23981.509,E2 -23981.509} C_VEL
LIN {X 0,Y 150.135,Z 376.78,A -85,B 0,C 180,E1 -23985.4,E2 -23985.4} C_VEL
LIN {X 0,Y 150.155,Z 376.779,A -85,B 0,C 180,E1 -23989.061,E2 -23989.061} C_VEL
LIN {X 0,Y 150.215,Z 376.771,A -85,B 0,C 180,E1 -23992.69,E2 -23992.69} C_VEL
LIN {X 0,Y 150.218,Z 376.771,A -85,B 0,C 180,E1 -23997.366,E2 -23997.366} C_VEL
LIN {X 0,Y 150.245,Z 376.763,A -85,B 0,C 180,E1 -24002.718,E2 -24002.718} C_VEL
LIN {X 0,Y 150.352,Z 376.755,A -85,B 0,C 180,E1 -24009.208,E2 -24009.208} C_VEL
LIN {X 0,Y 150.384,Z 376.752,A -85,B 0,C 180,E1 -24013.716,E2 -24013.716} C_VEL
LIN {X 0,Y 150.691,Z 376.71,A -85,B 0,C 180,E1 -24019.248,E2 -24019.248} C_VEL
LIN {X 0,Y 150.765,Z 376.706,A -85,B 0,C 180,E1 -24021.961,E2 -24021.961} C_VEL
LIN {X 0,Y 151.222,Z 376.648,A -85,B 0,C 180,E1 -24030,E2 -24030} C_VEL
LIN {X 0,Y 150.743,Z 376.708,A -85,B 0,C 180,E1 -24038.04,E2 -24038.04} C_VEL
LIN {X 0,Y 150.607,Z 376.72,A -85,B 0,C 180,E1 -24041.491,E2 -24041.491} C_VEL
LIN {X 0,Y 150.371,Z 376.752,A -85,B 0,C 180,E1 -24046.285,E2 -24046.285} C_VEL
LIN {X 0,Y 150.353,Z 376.755,A -85,B 0,C 180,E1 -24050.793,E2 -24050.793} C_VEL
LIN {X 0,Y 150.239,Z 376.771,A -85,B 0,C 180,E1 -24057.278,E2 -24057.278} C_VEL
LIN {X 0,Y 150.31,Z 376.936,A -85,B 0,C 180,E1 -24059.98,E2 -24059.98} C_VEL
LIN {X 0,Y 150.624,Z 378.134,A -85,B 0,C 180,E1 -24060.491,E2 -24060.491} C_VEL
LIN {X 0,Y 154.336,Z 390.531,A -85,B 0,C 180,E1 -24063.123,E2 -24063.123} C_VEL
LIN {X 0,Y 157.291,Z 401.747,A -85,B 0,C 180,E1 -24065.864,E2 -24065.864} C_VEL
LIN {X 0,Y 158.417,Z 406.459,A -85,B 0,C 180,E1 -24067.141,E2 -24067.141} C_VEL
LIN {X 0,Y 156.357,Z 417.688,A -85,B 0,C 180,E1 -24070.171,E2 -24070.171} C_VEL
LIN {X 0,Y 154.359,Z 428.259,A -85,B 0,C 180,E1 -24073.714,E2 -24073.714} C_VEL
LIN {X 0,Y 152.719,Z 437.089,A -85,B 0,C 180,E1 -24077.416,E2 -24077.416} C_VEL
LIN {X 0,Y 151.672,Z 444.066,A -85,B 0,C 180,E1 -24080.991,E2 -24080.991} C_VEL
LIN {X 0,Y 150.835,Z 450.788,A -85,B 0,C 180,E1 -24085.196,E2 -24085.196} C_VEL
LIN {X 0,Y 150.6,Z 455.855,A -85,B 0,C 180,E1 -24089.114,E2 -24089.114} C_VEL
LIN {X 0,Y 151.048,Z 460.647,A -85,B 0,C 180,E1 -24093.801,E2 -24093.801} C_VEL
LIN {X 0,Y 152.263,Z 464.046,A -85,B 0,C 180,E1 -24098.33,E2 -24098.33} C_VEL
